LIN {X 0,Y 363.033,Z 812.389,A -85,B 0,C 180,E1 -13571.073,E2 -13571.073} C_VEL
LIN {X 0,Y 362.364,Z 824.695,A -85,B 0,C 180,E1 -13571.915,E2 -13571.915} C_VEL
LIN {X 0,Y 361.562,Z 836.062,A -85,B 0,C 180,E1 -13572.935,E2 -13572.935} C_VEL
LIN {X 0,Y 360.7,Z 845.735,A -85,B 0,C 180,E1 -13574.019,E2 -13574.019} C_VEL
LIN {X 0,Y 359.815,Z 854.935,A -85,B 0,C 180,E1 -13575.284,E2 -13575.284} C_VEL
LIN {X 0,Y 358.912,Z 863.313,A -85,B 0,C 180,E1 -13576.691,E2 -13576.691} C_VEL
LIN {X 0,Y 357.851,Z 871.446,A -85,B 0,C 180,E1 -13578.38,E2 -13578.38} C_VEL
LIN {X 0,Y 357.002,Z 878.309,A -85,B 0,C 180,E1 -13580.172,E2 -13580.172} C_VEL
LIN {X 0,Y 356.417,Z 883.932,A -85,B 0,C 180,E1 -13582.059,E2 -13582.059} C_VEL
LIN {X 0,Y 355.754,Z 887.827,A -85,B 0,C 180,E1 -13583.755,E2 -13583.755} C_VEL
LIN {X 0,Y 355.31,Z 890.694,A -85,B 0,C 180,E1 -13585.455,E2 -13585.455} C_VEL
LIN {X 0,Y 355.23,Z 892.053,A -85,B 0,C 180,E1 -13586.59,E2 -13586.59} C_VEL
LIN {X 0,Y 355.216,Z 893.011,A -85,B 0,C 180,E1 -13587.725,E2 -13587.725} C_VEL
LIN {X 0,Y 355.044,Z 893.855,A -85,B 0,C 180,E1 -13589.992,E2 -13589.992} C_VEL
LIN {X 0,Y 355.224,Z 893.093,A -85,B 0,C 180,E1 -13592.26,E2 -13592.26} C_VEL
LIN {X 0,Y 355.295,Z 890.863,A -85,B 0,C 180,E1 -13594.53,E2 -13594.53} C_VEL
LIN {X 0,Y 355.742,Z 888.05,A -85,B 0,C 180,E1 -13596.23,E2 -13596.23} C_VEL
LIN {X 0,Y 356.389,Z 884.226,A -85,B 0,C 180,E1 -13597.926,E2 -13597.926} C_VEL
LIN {X 0,Y 356.975,Z 878.755,A -85,B 0,C 180,E1 -13599.803,E2 -13599.803} C_VEL
LIN {X 0,Y 357.831,Z 871.946,A -85,B 0,C 180,E1 -13601.605,E2 -13601.605} C_VEL
LIN {X 0,Y 358.881,Z 863.92,A -85,B 0,C 180,E1 -13603.294,E2 -13603.294} C_VEL
LIN {X 0,Y 359.776,Z 855.705,A -85,B 0,C 180,E1 -13604.702,E2 -13604.702} C_VEL
LIN {X 0,Y 360.732,Z 845.541,A -85,B 0,C 180,E1 -13606.11,E2 -13606.11} C_VEL
LIN {X 0,Y 361.701,Z 835.452,A -85,B 0,C 180,E1 -13607.226,E2 -13607.226} C_VEL
LIN {X 0,Y 361.408,Z 832.183,A -85,B 0,C 180,E1 -13607.582,E2 -13607.582} C_VEL
LIN {X 0,Y 359.137,Z 827.141,A -85,B 0,C 180,E1 -13608.205,E2 -13608.205} C_VEL
LIN {X 0,Y 356.76,Z 821.949,A -85,B 0,C 180,E1 -13608.788,E2 -13608.788} C_VEL
LIN {X 0,Y 356.293,Z 818.404,A -85,B 0,C 180,E1 -13609.072,E2 -13609.072} C_VEL
LIN {X 0,Y 356.661,Z 805.402,A -85,B 0,C 180,E1 -13609.825,E2 -13609.825} C_VEL
LIN {X 0,Y 356.867,Z 793.247,A -85,B 0,C 180,E1 -13610.301,E2 -13610.301} C_VEL
LIN {X 0,Y 357.103,Z 760.469,A -85,B 0,C 180,E1 -13611.017,E2 -13611.017} C_VEL
LIN {X 0,Y 357.565,Z 732.208,A -85,B 0,C 180,E1 -13611.588,E2 -13611.588} C_VEL
LIN {X 0,Y 348.581,Z 711.641,A -85,B 0,C 180,E1 -13612.655,E2 -13612.655} C_VEL
LIN {X 0,Y 347.782,Z 709.155,A -85,B 0,C 180,E1 -13612.804,E2 -13612.804} C_VEL
LIN {X 0,Y 347.806,Z 709.153,A -85,B 0,C 180,E1 -13616.384,E2 -13616.384} C_VEL
LIN {X 0,Y 347.721,Z 709.167,A -85,B 0,C 180,E1 -13620.339,E2 -13620.339} C_VEL
LIN {X 0,Y 347.716,Z 709.168,A -85,B 0,C 180,E1 -13624.035,E2 -13624.035} C_VEL
LIN {X 0,Y 347.727,Z 709.161,A -85,B 0,C 180,E1 -13627.312,E2 -13627.312} C_VEL
LIN {X 0,Y 347.754,Z 709.168,A -85,B 0,C 180,E1 -13630.28,E2 -13630.28} C_VEL
LIN {X 0,Y 347.777,Z 709.158,A -85,B 0,C 180,E1 -13633.385,E2 -13633.385} C_VEL
LIN {X 0,Y 347.772,Z 709.156,A -85,B 0,C 180,E1 -13636.663,E2 -13636.663} C_VEL
LIN {X 0,Y 347.737,Z 709.167,A -85,B 0,C 180,E1 -13640.158,E2 -13640.158} C_VEL
LIN {X 0,Y 347.735,Z 709.169,A -85,B 0,C 180,E1 -13644.118,E2 -13644.118} C_VEL
LIN {X 0,Y 347.706,Z 709.173,A -85,B 0,C 180,E1 -13648.296,E2 -13648.296} C_VEL
LIN {X 0,Y 347.746,Z 709.157,A -85,B 0,C 180,E1 -13650.984,E2 -13650.984} C_VEL
LIN {X 0,Y 347.77,Z 709.163,A -85,B 0,C 180,E1 -13653.603,E2 -13653.603} C_VEL
LIN {X 0,Y 347.725,Z 709.163,A -85,B 0,C 180,E1 -13656.157,E2 -13656.157} C_VEL
LIN {X 0,Y 347.747,Z 709.167,A -85,B 0,C 180,E1 -13659.905,E2 -13659.905} C_VEL
LIN {X 0,Y 347.8,Z 709.152,A -85,B 0,C 180,E1 -13662.356,E2 -13662.356} C_VEL
LIN {X 0,Y 347.83,Z 709.157,A -85,B 0,C 180,E1 -13665.968,E2 -13665.968} C_VEL
LIN {X 0,Y 347.864,Z 709.142,A -85,B 0,C 180,E1 -13669.524,E2 -13669.524} C_VEL
LIN {X 0,Y 348.026,Z 709.136,A -85,B 0,C 180,E1 -13673.041,E2 -13673.041} C_VEL
LIN {X 0,Y 348.145,Z 709.117,A -85,B 0,C 180,E1 -13677.686,E2 -13677.686} C_VEL
LIN {X 0,Y 348.297,Z 709.1,A -85,B 0,C 180,E1 -13680,E2 -13680} C_VEL
LIN {X 0,Y 348.145,Z 709.112,A -85,B 0,C 180,E1 -13682.314,E2 -13682.314} C_VEL
LIN {X 0,Y 348.025,Z 709.138,A -85,B 0,C 180,E1 -13686.959,E2 -13686.959} C_VEL
LIN {X 0,Y 347.864,Z 709.148,A -85,B 0,C 180,E1 -13690.476,E2 -13690.476} C_VEL
LIN {X 0,Y 347.831,Z 709.155,A -85,B 0,C 180,E1 -13694.153,E2 -13694.153} C_VEL
LIN {X 0,Y 347.824,Z 709.156,A -85,B 0,C 180,E1 -13698.293,E2 -13698.293} C_VEL
LIN {X 0,Y 347.712,Z 709.164,A -85,B 0,C 180,E1 -13701.634,E2 -13701.634} C_VEL
LIN {X 0,Y 347.75,Z 709.163,A -85,B 0,C 180,E1 -13705.113,E2 -13705.113} C_VEL
LIN {X 0,Y 347.752,Z 709.166,A -85,B 0,C 180,E1 -13707.699,E2 -13707.699} C_VEL
LIN {X 0,Y 347.712,Z 709.165,A -85,B 0,C 180,E1 -13710.352,E2 -13710.352} C_VEL
LIN {X 0,Y 347.693,Z 709.171,A -85,B 0,C 180,E1 -13714.05,E2 -13714.05} C_VEL
LIN {X 0,Y 347.714,Z 709.168,A -85,B 0,C 180,E1 -13717.327,E2 -13717.327} C_VEL
LIN {X 0,Y 347.744,Z 709.161,A -85,B 0,C 180,E1 -13720.296,E2 -13720.296} C_VEL
LIN {X 0,Y 347.773,Z 709.164,A -85,B 0,C 180,E1 -13723.401,E2 -13723.401} C_VEL
LIN {X 0,Y 347.775,Z 709.16,A -85,B 0,C 180,E1 -13726.678,E2 -13726.678} C_VEL
LIN {X 0,Y 347.747,Z 709.166,A -85,B 0,C 180,E1 -13730.173,E2 -13730.173} C_VEL
LIN {X 0,Y 347.742,Z 709.238,A -85,B 0,C 180,E1 -13733.578,E2 -13733.578} C_VEL
LIN {X 0,Y 350.722,Z 720.967,A -85,B 0,C 180,E1 -13736.217,E2 -13736.217} C_VEL
LIN {X 0,Y 354.282,Z 737.106,A -85,B 0,C 180,E1 -13739.623,E2 -13739.623} C_VEL
LIN {X 0,Y 354.467,Z 740.581,A -85,B 0,C 180,E1 -13740.297,E2 -13740.297} C_VEL
LIN {X 0,Y 351.936,Z 764.083,A -85,B 0,C 180,E1 -13744.584,E2 -13744.584} C_VEL
LIN {X 0,Y 350.688,Z 776.95,A -85,B 0,C 180,E1 -13746.947,E2 -13746.947} C_VEL
LIN {X 0,Y 354.861,Z 812.933,A -85,B 0,C 180,E1 -13747.995,E2 -13747.995} C_VEL
LIN {X 0,Y 356.332,Z 830.994,A -85,B 0,C 180,E1 -13748.467,E2 -13748.467} C_VEL
LIN {X 0,Y 355.113,Z 888.22,A -85,B 0,C 180,E1 -13749.633,E2 -13749.633} C_VEL
LIN {X 0,Y 354.393,Z 902.169,A -85,B 0,C 180,E1 -13750.156,E2 -13750.156} C_VEL
LIN {X 0,Y 353.32,Z 914.672,A -85,B 0,C 180,E1 -13750.849,E2 -13750.849} C_VEL
LIN {X 0,Y 352.199,Z 925.867,A -85,B 0,C 180,E1 -13751.692,E2 -13751.692} C_VEL
LIN {X 0,Y 350.897,Z 937.551,A -85,B 0,C 180,E1 -13752.826,E2 -13752.826} C_VEL
LIN {X 0,Y 349.706,Z 948.114,A -85,B 0,C 180,E1 -13754.117,E2 -13754.117} C_VEL
LIN {X 0,Y 348.615,Z 957.541,A -85,B 0,C 180,E1 -13755.542,E2 -13755.542} C_VEL
LIN {X 0,Y 348.169,Z 963.316,A -85,B 0,C 180,E1 -13756.586,E2 -13756.586} C_VEL
LIN {X 0,Y 347.394,Z 971.527,A -85,B 0,C 180,E1 -13758.337,E2 -13758.337} C_VEL
LIN {X 0,Y 346.965,Z 978.154,A -85,B 0,C 180,E1 -13760.094,E2 -13760.094} C_VEL
LIN {X 0,Y 346.829,Z 983.454,A -85,B 0,C 180,E1 -13761.854,E2 -13761.854} C_VEL
LIN {X 0,Y 346.912,Z 987.231,A -85,B 0,C 180,E1 -13763.433,E2 -13763.433} C_VEL
LIN {X 0,Y 347.049,Z 990.682,A -85,B 0,C 180,E1 -13765.362,E2 -13765.362} C_VEL
LIN {X 0,Y 347.141,Z 992.149,A -85,B 0,C 180,E1 -13766.526,E2 -13766.526} C_VEL
LIN {X 0,Y 347.188,Z 993.192,A -85,B 0,C 180,E1 -13767.688,E2 -13767.688} C_VEL
LIN {X 0,Y 347.262,Z 993.833,A -85,B 0,C 180,E1 -13768.848,E2 -13768.848} C_VEL
LIN {X 0,Y 347.327,Z 994.062,A -85,B 0,C 180,E1 -13770.008,E2 -13770.008} C_VEL
LIN {X 0,Y 347.263,Z 993.822,A -85,B 0,C 180,E1 -13771.167,E2 -13771.167} C_VEL
LIN {X 0,Y 347.19,Z 993.173,A -85,B 0,C 180,E1 -13772.328,E2 -13772.328} C_VEL
LIN {X 0,Y 347.144,Z 992.122,A -85,B 0,C 180,E1 -13773.489,E2 -13773.489} C_VEL
LIN {X 0,Y 347.05,Z 990.643,A -85,B 0,C 180,E1 -13774.654,E2 -13774.654} C_VEL
LIN {X 0,Y 346.834,Z 986.62,A -85,B 0,C 180,E1 -13776.829,E2 -13776.829} C_VEL
LIN {X 0,Y 346.85,Z 981.728,A -85,B 0,C 180,E1 -13778.748,E2 -13778.748} C_VEL
LIN {X 0,Y 347.072,Z 975.988,A -85,B 0,C 180,E1 -13780.508,E2 -13780.508} C_VEL
LIN {X 0,Y 347.604,Z 968.877,A -85,B 0,C 180,E1 -13782.264,E2 -13782.264} C_VEL
LIN {X 0,Y 348.419,Z 960.016,A -85,B 0,C 180,E1 -13784.015,E2 -13784.015} C_VEL
LIN {X 0,Y 349.011,Z 954.446,A -85,B 0,C 180,E1 -13784.943,E2 -13784.943} C_VEL
LIN {X 0,Y 349.854,Z 945.728,A -85,B 0,C 180,E1 -13786.191,E2 -13786.191} C_VEL
LIN {X 0,Y 351.166,Z 934.653,A -85,B 0,C 180,E1 -13787.476,E2 -13787.476} C_VEL
LIN {X 0,Y 352.408,Z 923.864,A -85,B 0,C 180,E1 -13788.464,E2 -13788.464} C_VEL
LIN {X 0,Y 354.182,Z 906.155,A -85,B 0,C 180,E1 -13789.721,E2 -13789.721} C_VEL
LIN {X 0,Y 355.294,Z 895.091,A -85,B 0,C 180,E1 -13790.335,E2 -13790.335} C_VEL
LIN {X 0,Y 356.158,Z 883.683,A -85,B 0,C 180,E1 -13790.812,E2 -13790.812} C_VEL
LIN {X 0,Y 358.768,Z 828.38,A -85,B 0,C 180,E1 -13792.478,E2 -13792.478} C_VEL
LIN {X 0,Y 357.212,Z 800.501,A -85,B 0,C 180,E1 -13793.658,E2 -13793.658} C_VEL
LIN {X 0,Y 354.765,Z 779.754,A -85,B 0,C 180,E1 -13794.75,E2 -13794.75} C_VEL
LIN {X 0,Y 352.506,Z 764.919,A -85,B 0,C 180,E1 -13795.644,E2 -13795.644} C_VEL
LIN {X 0,Y 352.154,Z 761.628,A -85,B 0,C 180,E1 -13795.852,E2 -13795.852} C_VEL
LIN {X 0,Y 354.226,Z 742.379,A -85,B 0,C 180,E1 -13799.362,E2 -13799.362} C_VEL
LIN {X 0,Y 354.422,Z 738.666,A -85,B 0,C 180,E1 -13800.052,E2 -13800.052} C_VEL
LIN {X 0,Y 352.311,Z 727.989,A -85,B 0,C 180,E1 -13802.256,E2 -13802.256} C_VEL
LIN {X 0,Y 348.952,Z 714.025,A -85,B 0,C 180,E1 -13805.305,E2 -13805.305} C_VEL
LIN {X 0,Y 347.756,Z 709.154,A -85,B 0,C 180,E1 -13806.471,E2 -13806.471} C_VEL
LIN {X 0,Y 347.72,Z 709.172,A -85,B 0,C 180,E1 -13809.821,E2 -13809.821} C_VEL
LIN {X 0,Y 347.732,Z 709.172,A -85,B 0,C 180,E1 -13813.413,E2 -13813.413} C_VEL
LIN {X 0,Y 347.74,Z 709.166,A -85,B 0,C 180,E1 -13816.691,E2 -13816.691} C_VEL
LIN {X 0,Y 347.721,Z 709.17,A -85,B 0,C 180,E1 -13820.185,E2 -13820.185} C_VEL
LIN {X 0,Y 347.774,Z 709.162,A -85,B 0,C 180,E1 -13822.681,E2 -13822.681} C_VEL
LIN {X 0,Y 347.769,Z 709.164,A -85,B 0,C 180,E1 -13825.959,E2 -13825.959} C_VEL
LIN {X 0,Y 347.756,Z 709.167,A -85,B 0,C 180,E1 -13829.653,E2 -13829.653} C_VEL
LIN {X 0,Y 347.781,Z 709.266,A -85,B 0,C 180,E1 -13833.721,E2 -13833.721} C_VEL
LIN {X 0,Y 348.906,Z 712.205,A -85,B 0,C 180,E1 -13834.053,E2 -13834.053} C_VEL
LIN {X 0,Y 350.729,Z 714.546,A -85,B 0,C 180,E1 -13834.467,E2 -13834.467} C_VEL
LIN {X 0,Y 352.786,Z 717.784,A -85,B 0,C 180,E1 -13834.933,E2 -13834.933} C_VEL
LIN {X 0,Y 358.789,Z 728.477,A -85,B 0,C 180,E1 -13836.248,E2 -13836.248} C_VEL
LIN {X 0,Y 362.716,Z 736.606,A -85,B 0,C 180,E1 -13837.071,E2 -13837.071} C_VEL
LIN {X 0,Y 359.911,Z 789.103,A -85,B 0,C 180,E1 -13838.71,E2 -13838.71} C_VEL
LIN {X 0,Y 359.641,Z 803.34,A -85,B 0,C 180,E1 -13839.256,E2 -13839.256} C_VEL
LIN {X 0,Y 359.183,Z 814.12,A -85,B 0,C 180,E1 -13839.814,E2 -13839.814} C_VEL
LIN {X 0,Y 358.405,Z 827.548,A -85,B 0,C 180,E1 -13840.736,E2 -13840.736} C_VEL
LIN {X 0,Y 357.419,Z 839.218,A -85,B 0,C 180,E1 -13841.811,E2 -13841.811} C_VEL
LIN {X 0,Y 356.472,Z 848.007,A -85,B 0,C 180,E1 -13842.799,E2 -13842.799} C_VEL
LIN {X 0,Y 355.531,Z 856.33,A -85,B 0,C 180,E1 -13843.934,E2 -13843.934} C_VEL
LIN {X 0,Y 354.571,Z 863.373,A -85,B 0,C 180,E1 -13845.068,E2 -13845.068} C_VEL
LIN {X 0,Y 353.694,Z 869.433,A -85,B 0,C 180,E1 -13846.205,E2 -13846.205} C_VEL
LIN {X 0,Y 352.613,Z 876.291,A -85,B 0,C 180,E1 -13847.775,E2 -13847.775} C_VEL
LIN {X 0,Y 351.765,Z 880.973,A -85,B 0,C 180,E1 -13849.059,E2 -13849.059} C_VEL
LIN {X 0,Y 350.8,Z 885.918,A -85,B 0,C 180,E1 -13850.777,E2 -13850.777} C_VEL
LIN {X 0,Y 349.947,Z 889.668,A -85,B 0,C 180,E1 -13852.499,E2 -13852.499} C_VEL
LIN {X 0,Y 349.298,Z 892.334,A -85,B 0,C 180,E1 -13854.226,E2 -13854.226} C_VEL
LIN {X 0,Y 349.029,Z 893.606,A -85,B 0,C 180,E1 -13855.38,E2 -13855.38} C_VEL
LIN {X 0,Y 348.461,Z 894.672,A -85,B 0,C 180,E1 -13857.688,E2 -13857.688} C_VEL
LIN {X 0,Y 348.268,Z 894.566,A -85,B 0,C 180,E1 -13858.844,E2 -13858.844} C_VEL
LIN {X 0,Y 348.031,Z 894.004,A -85,B 0,C 180,E1 -13860,E2 -13860} C_VEL
LIN {X 0,Y 347.875,Z 891.603,A -85,B 0,C 180,E1 -13862.316,E2 -13862.316} C_VEL
LIN {X 0,Y 347.823,Z 888.615,A -85,B 0,C 180,E1 -13864.055,E2 -13864.055} C_VEL
LIN {X 0,Y 348.192,Z 884.49,A -85,B 0,C 180,E1 -13865.792,E2 -13865.792} C_VEL
LIN {X 0,Y 348.488,Z 879.178,A -85,B 0,C 180,E1 -13867.532,E2 -13867.532} C_VEL
LIN {X 0,Y 348.81,Z 873.146,A -85,B 0,C 180,E1 -13869.127,E2 -13869.127} C_VEL
LIN {X 0,Y 349.155,Z 867.226,A -85,B 0,C 180,E1 -13870.437,E2 -13870.437} C_VEL
LIN {X 0,Y 349.647,Z 859.367,A -85,B 0,C 180,E1 -13871.89,E2 -13871.89} C_VEL
LIN {X 0,Y 350.099,Z 850.899,A -85,B 0,C 180,E1 -13873.2,E2 -13873.2} C_VEL
LIN {X 0,Y 350.606,Z 841.924,A -85,B 0,C 180,E1 -13874.363,E2 -13874.363} C_VEL
LIN {X 0,Y 351.081,Z 834.019,A -85,B 0,C 180,E1 -13875.233,E2 -13875.233} C_VEL
LIN {X 0,Y 351.558,Z 823.838,A -85,B 0,C 180,E1 -13876.169,E2 -13876.169} C_VEL
LIN {X 0,Y 351.952,Z 813.596,A -85,B 0,C 180,E1 -13876.935,E2 -13876.935} C_VEL
LIN {X 0,Y 352.228,Z 803.005,A -85,B 0,C 180,E1 -13877.565,E2 -13877.565} C_VEL
LIN {X 0,Y 352.457,Z 792.447,A -85,B 0,C 180,E1 -13878.041,E2 -13878.041} C_VEL
LIN {X 0,Y 352.627,Z 778.382,A -85,B 0,C 180,E1 -13878.483,E2 -13878.483} C_VEL
LIN {X 0,Y 353.651,Z 727.317,A -85,B 0,C 180,E1 -13879.826,E2 -13879.826} C_VEL
LIN {X 0,Y 347.832,Z 709.16,A -85,B 0,C 180,E1 -13880.594,E2 -13880.594} C_VEL
LIN {X 0,Y 347.824,Z 709.16,A -85,B 0,C 180,E1 -13884.588,E2 -13884.588} C_VEL
LIN {X 0,Y 347.757,Z 709.162,A -85,B 0,C 180,E1 -13887.699,E2 -13887.699} C_VEL
LIN {X 0,Y 347.757,Z 709.166,A -85,B 0,C 180,E1 -13890.347,E2 -13890.347} C_VEL
LIN {X 0,Y 347.77,Z 709.161,A -85,B 0,C 180,E1 -13894.041,E2 -13894.041} C_VEL
LIN {X 0,Y 347.775,Z 709.163,A -85,B 0,C 180,E1 -13897.319,E2 -13897.319} C_VEL
LIN {X 0,Y 347.717,Z 709.168,A -85,B 0,C 180,E1 -13900.299,E2 -13900.299} C_VEL
LIN {X 0,Y 347.741,Z 709.164,A -85,B 0,C 180,E1 -13903.406,E2 -13903.406} C_VEL
LIN {X 0,Y 347.743,Z 709.163,A -85,B 0,C 180,E1 -13906.684,E2 -13906.684} C_VEL
LIN {X 0,Y 347.721,Z 709.164,A -85,B 0,C 180,E1 -13910.179,E2 -13910.179} C_VEL
LIN {X 0,Y 347.773,Z 709.16,A -85,B 0,C 180,E1 -13912.674,E2 -13912.674} C_VEL
LIN {X 0,Y 347.767,Z 709.159,A -85,B 0,C 180,E1 -13915.952,E2 -13915.952} C_VEL
LIN {X 0,Y 347.744,Z 709.165,A -85,B 0,C 180,E1 -13919.645,E2 -13919.645} C_VEL
LIN {X 0,Y 347.748,Z 709.166,A -85,B 0,C 180,E1 -13923.594,E2 -13923.594} C_VEL
LIN {X 0,Y 347.799,Z 709.163,A -85,B 0,C 180,E1 -13927.337,E2 -13927.337} C_VEL
LIN {X 0,Y 348.822,Z 712.011,A -85,B 0,C 180,E1 -13927.479,E2 -13927.479} C_VEL
LIN {X 0,Y 357.48,Z 732.053,A -85,B 0,C 180,E1 -13928.51,E2 -13928.51} C_VEL
LIN {X 0,Y 356.849,Z 788.301,A -85,B 0,C 180,E1 -13929.67,E2 -13929.67} C_VEL
LIN {X 0,Y 356.776,Z 801.73,A -85,B 0,C 180,E1 -13930.117,E2 -13930.117} C_VEL
LIN {X 0,Y 356.395,Z 813.4,A -85,B 0,C 180,E1 -13930.706,E2 -13930.706} C_VEL
LIN {X 0,Y 355.69,Z 825.704,A -85,B 0,C 180,E1 -13931.564,E2 -13931.564} C_VEL
LIN {X 0,Y 354.849,Z 837.07,A -85,B 0,C 180,E1 -13932.602,E2 -13932.602} C_VEL
LIN {X 0,Y 353.949,Z 846.742,A -85,B 0,C 180,E1 -13933.705,E2 -13933.705} C_VEL
LIN {X 0,Y 353.023,Z 855.941,A -85,B 0,C 180,E1 -13934.994,E2 -13934.994} C_VEL
LIN {X 0,Y 352.076,Z 864.318,A -85,B 0,C 180,E1 -13936.428,E2 -13936.428} C_VEL
LIN {X 0,Y 350.971,Z 872.451,A -85,B 0,C 180,E1 -13938.149,E2 -13938.149} C_VEL
LIN {X 0,Y 350.079,Z 879.313,A -85,B 0,C 180,E1 -13939.976,E2 -13939.976} C_VEL
LIN {X 0,Y 349.459,Z 884.936,A -85,B 0,C 180,E1 -13941.9,E2 -13941.9} C_VEL
LIN {X 0,Y 348.77,Z 888.831,A -85,B 0,C 180,E1 -13943.63,E2 -13943.63} C_VEL
LIN {X 0,Y 348.304,Z 891.698,A -85,B 0,C 180,E1 -13945.363,E2 -13945.363} C_VEL
LIN {X 0,Y 348.215,Z 893.056,A -85,B 0,C 180,E1 -13946.521,E2 -13946.521} C_VEL
LIN {X 0,Y 348.196,Z 894.014,A -85,B 0,C 180,E1 -13947.679,E2 -13947.679} C_VEL
LIN {X 0,Y 348.017,Z 894.857,A -85,B 0,C 180,E1 -13949.992,E2 -13949.992} C_VEL
LIN {X 0,Y 348.203,Z 894.095,A -85,B 0,C 180,E1 -13952.306,E2 -13952.306} C_VEL
LIN {X 0,Y 348.288,Z 891.865,A -85,B 0,C 180,E1 -13954.622,E2 -13954.622} C_VEL
LIN {X 0,Y 348.758,Z 889.052,A -85,B 0,C 180,E1 -13956.355,E2 -13956.355} C_VEL
LIN {X 0,Y 349.433,Z 885.227,A -85,B 0,C 180,E1 -13958.085,E2 -13958.085} C_VEL
LIN {X 0,Y 350.052,Z 879.756,A -85,B 0,C 180,E1 -13959.999,E2 -13959.999} C_VEL
LIN {X 0,Y 350.95,Z 872.946,A -85,B 0,C 180,E1 -13961.836,E2 -13961.836} C_VEL
LIN {X 0,Y 352.047,Z 864.92,A -85,B 0,C 180,E1 -13963.557,E2 -13963.557} C_VEL
LIN {X 0,Y 352.982,Z 856.705,A -85,B 0,C 180,E1 -13964.992,E2 -13964.992} C_VEL
LIN {X 0,Y 353.987,Z 846.54,A -85,B 0,C 180,E1 -13966.425,E2 -13966.425} C_VEL
LIN {X 0,Y 355.045,Z 836.075,A -85,B 0,C 180,E1 -13967.599,E2 -13967.599} C_VEL
LIN {X 0,Y 355.858,Z 824.814,A -85,B 0,C 180,E1 -13968.609,E2 -13968.609} C_VEL
LIN {X 0,Y 356.293,Z 818.404,A -85,B 0,C 180,E1 -13969.072,E2 -13969.072} C_VEL
LIN {X 0,Y 355.976,Z 812.981,A -85,B 0,C 180,E1 -13969.452,E2 -13969.452} C_VEL
LIN {X 0,Y 352.445,Z 800.677,A -85,B 0,C 180,E1 -13970.321,E2 -13970.321} C_VEL
LIN {X 0,Y 350.683,Z 793.351,A -85,B 0,C 180,E1 -13970.703,E2 -13970.703} C_VEL
LIN {X 0,Y 350.349,Z 789.515,A -85,B 0,C 180,E1 -13970.827,E2 -13970.827} C_VEL
LIN {X 0,Y 350.766,Z 749.924,A -85,B 0,C 180,E1 -13971.665,E2 -13971.665} C_VEL
LIN {X 0,Y 351.042,Z 733.993,A -85,B 0,C 180,E1 -13971.992,E2 -13971.992} C_VEL
LIN {X 0,Y 341.602,Z 712.634,A -85,B 0,C 180,E1 -13973.146,E2 -13973.146} C_VEL
LIN {X 0,Y 340.745,Z 710.035,A -85,B 0,C 180,E1 -13973.302,E2 -13973.302} C_VEL
LIN {X 0,Y 340.779,Z 710.033,A -85,B 0,C 180,E1 -13976.971,E2 -13976.971} C_VEL
LIN {X 0,Y 340.669,Z 710.05,A -85,B 0,C 180,E1 -13981.036,E2 -13981.036} C_VEL
LIN {X 0,Y 340.685,Z 710.049,A -85,B 0,C 180,E1 -13985.27,E2 -13985.27} C_VEL
LIN {X 0,Y 340.676,Z 710.03,A -85,B 0,C 180,E1 -13988.378,E2 -13988.378} C_VEL
LIN {X 0,Y 340.685,Z 710.052,A -85,B 0,C 180,E1 -13991.296,E2 -13991.296} C_VEL
LIN {X 0,Y 340.738,Z 710.023,A -85,B 0,C 180,E1 -13994.515,E2 -13994.515} C_VEL
LIN {X 0,Y 340.705,Z 710.046,A -85,B 0,C 180,E1 -13997.937,E2 -13997.937} C_VEL
LIN {X 0,Y 340.684,Z 710.045,A -85,B 0,C 180,E1 -14000.245,E2 -14000.245} C_VEL
LIN {X 0,Y 340.658,Z 710.052,A -85,B 0,C 180,E1 -14003.553,E2 -14003.553} C_VEL
LIN {X 0,Y 340.64,Z 710.048,A -85,B 0,C 180,E1 -14006.147,E2 -14006.147} C_VEL
LIN {X 0,Y 340.717,Z 710.035,A -85,B 0,C 180,E1 -14010.327,E2 -14010.327} C_VEL
LIN {X 0,Y 340.744,Z 710.037,A -85,B 0,C 180,E1 -14013.015,E2 -14013.015} C_VEL
LIN {X 0,Y 340.665,Z 710.043,A -85,B 0,C 180,E1 -14016.922,E2 -14016.922} C_VEL
LIN {X 0,Y 340.725,Z 710.038,A -85,B 0,C 180,E1 -14020.73,E2 -14020.73} C_VEL
LIN {X 0,Y 340.72,Z 710.034,A -85,B 0,C 180,E1 -14023.215,E2 -14023.215} C_VEL
LIN {X 0,Y 340.778,Z 710.035,A -85,B 0,C 180,E1 -14026.888,E2 -14026.888} C_VEL
LIN {X 0,Y 340.859,Z 710.019,A -85,B 0,C 180,E1 -14030.506,E2 -14030.506} C_VEL
LIN {X 0,Y 340.993,Z 710.014,A -85,B 0,C 180,E1 -14032.896,E2 -14032.896} C_VEL
LIN {X 0,Y 341.108,Z 709.994,A -85,B 0,C 180,E1 -14037.638,E2 -14037.638} C_VEL
LIN {X 0,Y 341.246,Z 709.979,A -85,B 0,C 180,E1 -14040,E2 -14040} C_VEL
LIN {X 0,Y 341.108,Z 709.988,A -85,B 0,C 180,E1 -14042.362,E2 -14042.362} C_VEL
LIN {X 0,Y 340.993,Z 710.012,A -85,B 0,C 180,E1 -14047.103,E2 -14047.103} C_VEL
LIN {X 0,Y 340.806,Z 710.028,A -85,B 0,C 180,E1 -14050.696,E2 -14050.696} C_VEL
LIN {X 0,Y 340.796,Z 710.031,A -85,B 0,C 180,E1 -14054.328,E2 -14054.328} C_VEL
LIN {X 0,Y 340.771,Z 710.034,A -85,B 0,C 180,E1 -14058.469,E2 -14058.469} C_VEL
LIN {X 0,Y 340.659,Z 710.045,A -85,B 0,C 180,E1 -14061.848,E2 -14061.848} C_VEL
LIN {X 0,Y 340.711,Z 710.037,A -85,B 0,C 180,E1 -14065.669,E2 -14065.669} C_VEL
LIN {X 0,Y 340.682,Z 710.046,A -85,B 0,C 180,E1 -14068.325,E2 -14068.325} C_VEL
LIN {X 0,Y 340.658,Z 710.044,A -85,B 0,C 180,E1 -14071.049,E2 -14071.049} C_VEL
LIN {X 0,Y 340.664,Z 710.047,A -85,B 0,C 180,E1 -14075.285,E2 -14075.285} C_VEL
LIN {X 0,Y 340.663,Z 710.034,A -85,B 0,C 180,E1 -14078.394,E2 -14078.394} C_VEL
LIN {X 0,Y 340.677,Z 710.048,A -85,B 0,C 180,E1 -14081.311,E2 -14081.311} C_VEL
LIN {X 0,Y 340.736,Z 710.041,A -85,B 0,C 180,E1 -14084.53,E2 -14084.53} C_VEL
LIN {X 0,Y 340.71,Z 710.036,A -85,B 0,C 180,E1 -14087.953,E2 -14087.953} C_VEL
LIN {X 0,Y 340.695,Z 710.043,A -85,B 0,C 180,E1 -14090.26,E2 -14090.26} C_VEL
LIN {X 0,Y 340.698,Z 710.136,A -85,B 0,C 180,E1 -14093.109,E2 -14093.109} C_VEL
LIN {X 0,Y 344.101,Z 723.516,A -85,B 0,C 180,E1 -14096.194,E2 -14096.194} C_VEL
LIN {X 0,Y 347.263,Z 737.936,A -85,B 0,C 180,E1 -14099.307,E2 -14099.307} C_VEL
LIN {X 0,Y 347.647,Z 740.989,A -85,B 0,C 180,E1 -14099.929,E2 -14099.929} C_VEL
LIN {X 0,Y 345.199,Z 763.104,A -85,B 0,C 180,E1 -14104.058,E2 -14104.058} C_VEL
LIN {X 0,Y 343.868,Z 776.212,A -85,B 0,C 180,E1 -14106.478,E2 -14106.478} C_VEL
LIN {X 0,Y 347.914,Z 810.535,A -85,B 0,C 180,E1 -14107.502,E2 -14107.502} C_VEL
LIN {X 0,Y 349.706,Z 831.274,A -85,B 0,C 180,E1 -14108.065,E2 -14108.065} C_VEL
LIN {X 0,Y 348.435,Z 887.216,A -85,B 0,C 180,E1 -14109.224,E2 -14109.224} C_VEL
LIN {X 0,Y 347.781,Z 900.401,A -85,B 0,C 180,E1 -14109.724,E2 -14109.724} C_VEL
LIN {X 0,Y 346.647,Z 913.669,A -85,B 0,C 180,E1 -14110.466,E2 -14110.466} C_VEL
LIN {X 0,Y 345.443,Z 924.856,A -85,B 0,C 180,E1 -14111.32,E2 -14111.32} C_VEL
LIN {X 0,Y 344.084,Z 936.537,A -85,B 0,C 180,E1 -14112.475,E2 -14112.475} C_VEL
LIN {X 0,Y 342.778,Z 947.088,A -85,B 0,C 180,E1 -14113.788,E2 -14113.788} C_VEL
LIN {X 0,Y 341.778,Z 955.796,A -85,B 0,C 180,E1 -14115.12,E2 -14115.12} C_VEL
LIN {X 0,Y 341.247,Z 962.302,A -85,B 0,C 180,E1 -14116.309,E2 -14116.309} C_VEL
LIN {X 0,Y 340.394,Z 970.509,A -85,B 0,C 180,E1 -14118.093,E2 -14118.093} C_VEL
LIN {X 0,Y 339.918,Z 977.134,A -85,B 0,C 180,E1 -14119.887,E2 -14119.887} C_VEL
LIN {X 0,Y 339.758,Z 982.435,A -85,B 0,C 180,E1 -14121.683,E2 -14121.683} C_VEL
LIN {X 0,Y 339.829,Z 985.719,A -85,B 0,C 180,E1 -14123.068,E2 -14123.068} C_VEL
LIN {X 0,Y 339.992,Z 989.672,A -85,B 0,C 180,E1 -14125.265,E2 -14125.265} C_VEL
LIN {X 0,Y 340.096,Z 991.142,A -85,B 0,C 180,E1 -14126.454,E2 -14126.454} C_VEL
LIN {X 0,Y 340.145,Z 992.187,A -85,B 0,C 180,E1 -14127.64,E2 -14127.64} C_VEL
LIN {X 0,Y 340.226,Z 992.829,A -85,B 0,C 180,E1 -14128.824,E2 -14128.824} C_VEL
LIN {X 0,Y 340.297,Z 993.059,A -85,B 0,C 180,E1 -14130.008,E2 -14130.008} C_VEL
LIN {X 0,Y 340.226,Z 992.818,A -85,B 0,C 180,E1 -14131.191,E2 -14131.191} C_VEL
LIN {X 0,Y 340.147,Z 992.167,A -85,B 0,C 180,E1 -14132.376,E2 -14132.376} C_VEL
LIN {X 0,Y 340.099,Z 991.114,A -85,B 0,C 180,E1 -14133.562,E2 -14133.562} C_VEL
LIN {X 0,Y 339.991,Z 989.632,A -85,B 0,C 180,E1 -14134.75,E2 -14134.75} C_VEL
LIN {X 0,Y 339.777,Z 985.85,A -85,B 0,C 180,E1 -14136.859,E2 -14136.859} C_VEL
LIN {X 0,Y 339.799,Z 980.709,A -85,B 0,C 180,E1 -14138.931,E2 -14138.931} C_VEL
LIN {X 0,Y 340.012,Z 974.962,A -85,B 0,C 180,E1 -14140.728,E2 -14140.728} C_VEL
LIN {X 0,Y 340.597,Z 967.852,A -85,B 0,C 180,E1 -14142.52,E2 -14142.52} C_VEL
LIN {X 0,Y 341.342,Z 960.629,A -85,B 0,C 180,E1 -14144.007,E2 -14144.007} C_VEL
LIN {X 0,Y 341.669,Z 956.525,A -85,B 0,C 180,E1 -14144.746,E2 -14144.746} C_VEL
LIN {X 0,Y 342.727,Z 947.967,A -85,B 0,C 180,E1 -14146.078,E2 -14146.078} C_VEL
LIN {X 0,Y 343.914,Z 937.592,A -85,B 0,C 180,E1 -14147.396,E2 -14147.396} C_VEL
LIN {X 0,Y 345.657,Z 923.215,A -85,B 0,C 180,E1 -14148.838,E2 -14148.838} C_VEL
LIN {X 0,Y 346.914,Z 913.267,A -85,B 0,C 180,E1 -14149.689,E2 -14149.689} C_VEL
LIN {X 0,Y 348.062,Z 903.107,A -85,B 0,C 180,E1 -14150.391,E2 -14150.391} C_VEL
LIN {X 0,Y 349.241,Z 891.716,A -85,B 0,C 180,E1 -14151.012,E2 -14151.012} C_VEL
LIN {X 0,Y 350.096,Z 880.865,A -85,B 0,C 180,E1 -14151.459,E2 -14151.459} C_VEL
LIN {X 0,Y 352.68,Z 828.91,A -85,B 0,C 180,E1 -14153.081,E2 -14153.081} C_VEL
LIN {X 0,Y 351.318,Z 801.407,A -85,B 0,C 180,E1 -14154.3,E2 -14154.3} C_VEL
LIN {X 0,Y 349.158,Z 781.767,A -85,B 0,C 180,E1 -14155.378,E2 -14155.378} C_VEL
LIN {X 0,Y 346.526,Z 763.396,A -85,B 0,C 180,E1 -14156.538,E2 -14156.538} C_VEL
LIN {X 0,Y 345.726,Z 757.568,A -85,B 0,C 180,E1 -14156.963,E2 -14156.963} C_VEL
LIN {X 0,Y 347.567,Z 740.712,A -85,B 0,C 180,E1 -14160.113,E2 -14160.113} C_VEL
LIN {X 0,Y 345.641,Z 730.447,A -85,B 0,C 180,E1 -14162.266,E2 -14162.266} C_VEL
LIN {X 0,Y 342.372,Z 716.624,A -85,B 0,C 180,E1 -14165.348,E2 -14165.348} C_VEL
LIN {X 0,Y 340.716,Z 710.035,A -85,B 0,C 180,E1 -14166.932,E2 -14166.932} C_VEL
LIN {X 0,Y 340.669,Z 710.048,A -85,B 0,C 180,E1 -14170.243,E2 -14170.243} C_VEL
LIN {X 0,Y 340.662,Z 710.05,A -85,B 0,C 180,E1 -14173.775,E2 -14173.775} C_VEL
LIN {X 0,Y 340.684,Z 710.047,A -85,B 0,C 180,E1 -14177.097,E2 -14177.097} C_VEL
LIN {X 0,Y 340.675,Z 710.047,A -85,B 0,C 180,E1 -14180.244,E2 -14180.244} C_VEL
LIN {X 0,Y 340.727,Z 710.045,A -85,B 0,C 180,E1 -14183.563,E2 -14183.563} C_VEL
LIN {X 0,Y 340.711,Z 710.042,A -85,B 0,C 180,E1 -14186.155,E2 -14186.155} C_VEL
LIN {X 0,Y 340.74,Z 710.04,A -85,B 0,C 180,E1 -14190.038,E2 -14190.038} C_VEL
LIN {X 0,Y 340.754,Z 710.246,A -85,B 0,C 180,E1 -14192.492,E2 -14192.492} C_VEL
LIN {X 0,Y 341.762,Z 712.908,A -85,B 0,C 180,E1 -14192.83,E2 -14192.83} C_VEL
LIN {X 0,Y 343.792,Z 715.402,A -85,B 0,C 180,E1 -14193.347,E2 -14193.347} C_VEL
LIN {X 0,Y 345.708,Z 718.547,A -85,B 0,C 180,E1 -14193.83,E2 -14193.83} C_VEL
LIN {X 0,Y 350.832,Z 726.883,A -85,B 0,C 180,E1 -14195.057,E2 -14195.057} C_VEL
LIN {X 0,Y 356.547,Z 738.013,A -85,B 0,C 180,E1 -14196.353,E2 -14196.353} C_VEL
LIN {X 0,Y 356.969,Z 739.093,A -85,B 0,C 180,E1 -14196.452,E2 -14196.452} C_VEL
LIN {X 0,Y 353.976,Z 790.114,A -85,B 0,C 180,E1 -14198.106,E2 -14198.106} C_VEL
LIN {X 0,Y 353.666,Z 804.276,A -85,B 0,C 180,E1 -14198.66,E2 -14198.66} C_VEL
LIN {X 0,Y 353.269,Z 813.946,A -85,B 0,C 180,E1 -14199.159,E2 -14199.159} C_VEL
LIN {X 0,Y 352.675,Z 824.025,A -85,B 0,C 180,E1 -14199.827,E2 -14199.827} C_VEL
LIN {X 0,Y 352.002,Z 832.285,A -85,B 0,C 180,E1 -14200.493,E2 -14200.493} C_VEL
LIN {X 0,Y 351.207,Z 840.853,A -85,B 0,C 180,E1 -14201.326,E2 -14201.326} C_VEL
LIN {X 0,Y 350.173,Z 849.534,A -85,B 0,C 180,E1 -14202.328,E2 -14202.328} C_VEL
LIN {X 0,Y 349.315,Z 856.902,A -85,B 0,C 180,E1 -14203.339,E2 -14203.339} C_VEL
LIN {X 0,Y 348.316,Z 864.07,A -85,B 0,C 180,E1 -14204.494,E2 -14204.494} C_VEL
LIN {X 0,Y 347.104,Z 871.503,A -85,B 0,C 180,E1 -14205.938,E2 -14205.938} C_VEL
LIN {X 0,Y 346.031,Z 877.693,A -85,B 0,C 180,E1 -14207.407,E2 -14207.407} C_VEL
LIN {X 0,Y 345.026,Z 882.722,A -85,B 0,C 180,E1 -14208.842,E2 -14208.842} C_VEL
LIN {X 0,Y 344.412,Z 886.162,A -85,B 0,C 180,E1 -14210.012,E2 -14210.012} C_VEL
LIN {X 0,Y 343.374,Z 890.208,A -85,B 0,C 180,E1 -14211.763,E2 -14211.763} C_VEL
LIN {X 0,Y 342.765,Z 892.224,A -85,B 0,C 180,E1 -14212.933,E2 -14212.933} C_VEL
LIN {X 0,Y 342.087,Z 894.914,A -85,B 0,C 180,E1 -14215.286,E2 -14215.286} C_VEL
LIN {X 0,Y 341.483,Z 895.869,A -85,B 0,C 180,E1 -14217.641,E2 -14217.641} C_VEL
LIN {X 0,Y 341.283,Z 895.663,A -85,B 0,C 180,E1 -14218.82,E2 -14218.82} C_VEL
LIN {X 0,Y 341.008,Z 895.042,A -85,B 0,C 180,E1 -14220,E2 -14220} C_VEL
LIN {X 0,Y 340.848,Z 892.447,A -85,B 0,C 180,E1 -14222.364,E2 -14222.364} C_VEL
LIN {X 0,Y 340.8,Z 889.32,A -85,B 0,C 180,E1 -14224.139,E2 -14224.139} C_VEL
LIN {X 0,Y 341.15,Z 885.066,A -85,B 0,C 180,E1 -14225.912,E2 -14225.912} C_VEL
LIN {X 0,Y 341.418,Z 880.654,A -85,B 0,C 180,E1 -14227.392,E2 -14227.392} C_VEL
LIN {X 0,Y 341.696,Z 875.52,A -85,B 0,C 180,E1 -14228.823,E2 -14228.823} C_VEL
LIN {X 0,Y 342.054,Z 868.867,A -85,B 0,C 180,E1 -14230.357,E2 -14230.357} C_VEL
LIN {X 0,Y 342.549,Z 861.092,A -85,B 0,C 180,E1 -14231.839,E2 -14231.839} C_VEL
LIN {X 0,Y 343.02,Z 852.723,A -85,B 0,C 180,E1 -14233.176,E2 -14233.176} C_VEL
LIN {X 0,Y 343.501,Z 843.871,A -85,B 0,C 180,E1 -14234.364,E2 -14234.364} C_VEL
LIN {X 0,Y 344.084,Z 834.655,A -85,B 0,C 180,E1 -14235.398,E2 -14235.398} C_VEL
LIN {X 0,Y 344.508,Z 825.929,A -85,B 0,C 180,E1 -14236.226,E2 -14236.226} C_VEL
LIN {X 0,Y 344.962,Z 814.467,A -85,B 0,C 180,E1 -14237.106,E2 -14237.106} C_VEL
LIN {X 0,Y 345.242,Z 803.989,A -85,B 0,C 180,E1 -14237.741,E2 -14237.741} C_VEL
LIN {X 0,Y 345.489,Z 793.454,A -85,B 0,C 180,E1 -14238.226,E2 -14238.226} C_VEL
LIN {X 0,Y 345.635,Z 779.445,A -85,B 0,C 180,E1 -14238.678,E2 -14238.678} C_VEL
LIN {X 0,Y 346.676,Z 728.505,A -85,B 0,C 180,E1 -14240.055,E2 -14240.055} C_VEL
LIN {X 0,Y 340.763,Z 710.04,A -85,B 0,C 180,E1 -14240.839,E2 -14240.839} C_VEL
LIN {X 0,Y 340.759,Z 710.039,A -85,B 0,C 180,E1 -14244.831,E2 -14244.831} C_VEL
LIN {X 0,Y 340.704,Z 710.042,A -85,B 0,C 180,E1 -14248.323,E2 -14248.323} C_VEL
LIN {X 0,Y 340.712,Z 710.045,A -85,B 0,C 180,E1 -14251.043,E2 -14251.043} C_VEL
LIN {X 0,Y 340.736,Z 710.039,A -85,B 0,C 180,E1 -14255.277,E2 -14255.277} C_VEL
LIN {X 0,Y 340.714,Z 710.041,A -85,B 0,C 180,E1 -14258.379,E2 -14258.379} C_VEL
LIN {X 0,Y 340.711,Z 710.038,A -85,B 0,C 180,E1 -14262.04,E2 -14262.04} C_VEL
LIN {X 0,Y 340.67,Z 710.043,A -85,B 0,C 180,E1 -14266.224,E2 -14266.224} C_VEL
LIN {X 0,Y 340.688,Z 710.043,A -85,B 0,C 180,E1 -14268.684,E2 -14268.684} C_VEL
LIN {X 0,Y 340.738,Z 710.035,A -85,B 0,C 180,E1 -14271.766,E2 -14271.766} C_VEL
LIN {X 0,Y 340.741,Z 710.037,A -85,B 0,C 180,E1 -14275.592,E2 -14275.592} C_VEL
LIN {X 0,Y 340.699,Z 710.042,A -85,B 0,C 180,E1 -14278.949,E2 -14278.949} C_VEL
LIN {X 0,Y 340.725,Z 710.041,A -85,B 0,C 180,E1 -14283.006,E2 -14283.006} C_VEL
LIN {X 0,Y 340.735,Z 710.041,A -85,B 0,C 180,E1 -14286.827,E2 -14286.827} C_VEL
LIN {X 0,Y 341.729,Z 712.85,A -85,B 0,C 180,E1 -14286.979,E2 -14286.979} C_VEL
LIN {X 0,Y 350.762,Z 733.385,A -85,B 0,C 180,E1 -14288.084,E2 -14288.084} C_VEL
LIN {X 0,Y 350.973,Z 737.009,A -85,B 0,C 180,E1 -14288.177,E2 -14288.177} C_VEL
LIN {X 0,Y 350.253,Z 788.436,A -85,B 0,C 180,E1 -14289.247,E2 -14289.247} C_VEL
LIN {X 0,Y 350.169,Z 802.04,A -85,B 0,C 180,E1 -14289.696,E2 -14289.696} C_VEL
LIN {X 0,Y 349.767,Z 814.412,A -85,B 0,C 180,E1 -14290.326,E2 -14290.326} C_VEL
LIN {X 0,Y 349.03,Z 826.713,A -85,B 0,C 180,E1 -14291.199,E2 -14291.199} C_VEL
LIN {X 0,Y 348.15,Z 838.077,A -85,B 0,C 180,E1 -14292.256,E2 -14292.256} C_VEL
LIN {X 0,Y 347.209,Z 847.748,A -85,B 0,C 180,E1 -14293.38,E2 -14293.38} C_VEL
LIN {X 0,Y 346.24,Z 856.947,A -85,B 0,C 180,E1 -14294.693,E2 -14294.693} C_VEL
LIN {X 0,Y 345.249,Z 865.323,A -85,B 0,C 180,E1 -14296.154,E2 -14296.154} C_VEL
LIN {X 0,Y 344.096,Z 873.456,A -85,B 0,C 180,E1 -14297.909,E2 -14297.909} C_VEL
LIN {X 0,Y 343.161,Z 880.318,A -85,B 0,C 180,E1 -14299.771,E2 -14299.771} C_VEL
LIN {X 0,Y 342.504,Z 885.94,A -85,B 0,C 180,E1 -14301.734,E2 -14301.734} C_VEL
LIN {X 0,Y 341.787,Z 889.834,A -85,B 0,C 180,E1 -14303.499,E2 -14303.499} C_VEL
LIN {X 0,Y 341.299,Z 892.701,A -85,B 0,C 180,E1 -14305.268,E2 -14305.268} C_VEL
LIN {X 0,Y 341.2,Z 894.059,A -85,B 0,C 180,E1 -14306.45,E2 -14306.45} C_VEL
LIN {X 0,Y 341.177,Z 895.017,A -85,B 0,C 180,E1 -14307.631,E2 -14307.631} C_VEL
LIN {X 0,Y 340.991,Z 895.859,A -85,B 0,C 180,E1 -14309.992,E2 -14309.992} C_VEL
LIN {X 0,Y 341.182,Z 895.097,A -85,B 0,C 180,E1 -14312.353,E2 -14312.353} C_VEL
LIN {X 0,Y 341.283,Z 892.867,A -85,B 0,C 180,E1 -14314.717,E2 -14314.717} C_VEL
LIN {X 0,Y 341.775,Z 890.054,A -85,B 0,C 180,E1 -14316.486,E2 -14316.486} C_VEL
LIN {X 0,Y 342.479,Z 886.228,A -85,B 0,C 180,E1 -14318.25,E2 -14318.25} C_VEL
LIN {X 0,Y 343.133,Z 880.757,A -85,B 0,C 180,E1 -14320.203,E2 -14320.203} C_VEL
LIN {X 0,Y 344.075,Z 873.947,A -85,B 0,C 180,E1 -14322.076,E2 -14322.076} C_VEL
LIN {X 0,Y 345.22,Z 865.92,A -85,B 0,C 180,E1 -14323.831,E2 -14323.831} C_VEL
LIN {X 0,Y 346.198,Z 857.704,A -85,B 0,C 180,E1 -14325.293,E2 -14325.293} C_VEL
LIN {X 0,Y 347.253,Z 847.538,A -85,B 0,C 180,E1 -14326.753,E2 -14326.753} C_VEL
LIN {X 0,Y 348.349,Z 837.075,A -85,B 0,C 180,E1 -14327.948,E2 -14327.948} C_VEL
LIN {X 0,Y 349.247,Z 825.284,A -85,B 0,C 180,E1 -14329.02,E2 -14329.02} C_VEL
LIN {X 0,Y 349.913,Z 812.748,A -85,B 0,C 180,E1 -14329.871,E2 -14329.871} C_VEL
LIN {X 0,Y 350.246,Z 800.519,A -85,B 0,C 180,E1 -14330.471,E2 -14330.471} C_VEL
LIN {X 0,Y 350.349,Z 789.515,A -85,B 0,C 180,E1 -14330.827,E2 -14330.827} C_VEL
LIN {X 0,Y 349.729,Z 783.743,A -85,B 0,C 180,E1 -14331.009,E2 -14331.009} C_VEL
LIN {X 0,Y 344.535,Z 765.174,A -85,B 0,C 180,E1 -14331.763,E2 -14331.763} C_VEL
LIN {X 0,Y 344.041,Z 759.382,A -85,B 0,C 180,E1 -14331.922,E2 -14331.922} C_VEL
LIN {X 0,Y 344.441,Z 735.635,A -85,B 0,C 180,E1 -14332.422,E2 -14332.422} C_VEL
LIN {X 0,Y 334.871,Z 714.04,A -85,B 0,C 180,E1 -14333.63,E2 -14333.63} C_VEL
LIN {X 0,Y 333.74,Z 711.169,A -85,B 0,C 180,E1 -14333.786,E2 -14333.786} C_VEL
LIN {X 0,Y 333.695,Z 710.914,A -85,B 0,C 180,E1 -14333.907,E2 -14333.907} C_VEL
LIN {X 0,Y 333.714,Z 710.91,A -85,B 0,C 180,E1 -14337.59,E2 -14337.59} C_VEL
LIN {X 0,Y 333.662,Z 710.919,A -85,B 0,C 180,E1 -14340.354,E2 -14340.354} C_VEL
LIN {X 0,Y 333.641,Z 710.921,A -85,B 0,C 180,E1 -14344.65,E2 -14344.65} C_VEL
LIN {X 0,Y 333.618,Z 710.913,A -85,B 0,C 180,E1 -14347.642,E2 -14347.642} C_VEL
LIN {X 0,Y 333.66,Z 710.924,A -85,B 0,C 180,E1 -14350.751,E2 -14350.751} C_VEL
LIN {X 0,Y 333.686,Z 710.903,A -85,B 0,C 180,E1 -14354.266,E2 -14354.266} C_VEL
LIN {X 0,Y 333.659,Z 710.92,A -85,B 0,C 180,E1 -14357.621,E2 -14357.621} C_VEL
LIN {X 0,Y 333.629,Z 710.922,A -85,B 0,C 180,E1 -14361.189,E2 -14361.189} C_VEL
LIN {X 0,Y 333.631,Z 710.922,A -85,B 0,C 180,E1 -14365.22,E2 -14365.22} C_VEL
LIN {X 0,Y 333.588,Z 710.933,A -85,B 0,C 180,E1 -14368.217,E2 -14368.217} C_VEL
LIN {X 0,Y 333.652,Z 710.912,A -85,B 0,C 180,E1 -14371.022,E2 -14371.022} C_VEL
LIN {X 0,Y 333.674,Z 710.92,A -85,B 0,C 180,E1 -14373.748,E2 -14373.748} C_VEL
LIN {X 0,Y 333.657,Z 710.917,A -85,B 0,C 180,E1 -14377.91,E2 -14377.91} C_VEL
LIN {X 0,Y 333.728,Z 710.907,A -85,B 0,C 180,E1 -14381.586,E2 -14381.586} C_VEL
LIN {X 0,Y 333.742,Z 710.911,A -85,B 0,C 180,E1 -14385.574,E2 -14385.574} C_VEL
LIN {X 0,Y 333.769,Z 710.898,A -85,B 0,C 180,E1 -14389.076,E2 -14389.076} C_VEL
LIN {X 0,Y 333.945,Z 710.893,A -85,B 0,C 180,E1 -14392.746,E2 -14392.746} C_VEL
LIN {X 0,Y 333.751,Z 710.903,A -85,B 0,C 180,E1 -14395.168,E2 -14395.168} C_VEL
LIN {X 0,Y 334.07,Z 710.871,A -85,B 0,C 180,E1 -14397.588,E2 -14397.588} C_VEL
LIN {X 0,Y 334.197,Z 710.857,A -85,B 0,C 180,E1 -14400,E2 -14400} C_VEL
LIN {X 0,Y 334.07,Z 710.865,A -85,B 0,C 180,E1 -14402.411,E2 -14402.411} C_VEL
LIN {X 0,Y 333.945,Z 710.887,A -85,B 0,C 180,E1 -14407.254,E2 -14407.254} C_VEL
LIN {X 0,Y 333.769,Z 710.906,A -85,B 0,C 180,E1 -14410.924,E2 -14410.924} C_VEL
LIN {X 0,Y 333.742,Z 710.91,A -85,B 0,C 180,E1 -14414.637,E2 -14414.637} C_VEL
LIN {X 0,Y 333.73,Z 710.912,A -85,B 0,C 180,E1 -14418.658,E2 -14418.658} C_VEL
LIN {X 0,Y 333.598,Z 710.928,A -85,B 0,C 180,E1 -14422.285,E2 -14422.285} C_VEL
LIN {X 0,Y 333.675,Z 710.913,A -85,B 0,C 180,E1 -14426.251,E2 -14426.251} C_VEL
LIN {X 0,Y 333.653,Z 710.92,A -85,B 0,C 180,E1 -14428.978,E2 -14428.978} C_VEL
LIN {X 0,Y 333.595,Z 710.929,A -85,B 0,C 180,E1 -14432.595,E2 -14432.595} C_VEL
LIN {X 0,Y 333.624,Z 710.928,A -85,B 0,C 180,E1 -14436.146,E2 -14436.146} C_VEL
LIN {X 0,Y 333.633,Z 710.908,A -85,B 0,C 180,E1 -14439.194,E2 -14439.194} C_VEL
LIN {X 0,Y 333.656,Z 710.922,A -85,B 0,C 180,E1 -14442.521,E2 -14442.521} C_VEL
LIN {X 0,Y 333.686,Z 710.921,A -85,B 0,C 180,E1 -14445.985,E2 -14445.985} C_VEL
LIN {X 0,Y 333.662,Z 710.924,A -85,B 0,C 180,E1 -14449.313,E2 -14449.313} C_VEL
LIN {X 0,Y 333.68,Z 711.103,A -85,B 0,C 180,E1 -14452.636,E2 -14452.636} C_VEL
LIN {X 0,Y 337.048,Z 724.209,A -85,B 0,C 180,E1 -14455.749,E2 -14455.749} C_VEL
LIN {X 0,Y 340.522,Z 740.124,A -85,B 0,C 180,E1 -14459.271,E2 -14459.271} C_VEL
LIN {X 0,Y 340.686,Z 743.35,A -85,B 0,C 180,E1 -14459.927,E2 -14459.927} C_VEL
LIN {X 0,Y 338.068,Z 765.355,A -85,B 0,C 180,E1 -14464.126,E2 -14464.126} C_VEL
LIN {X 0,Y 337.08,Z 774.856,A -85,B 0,C 180,E1 -14465.956,E2 -14465.956} C_VEL
LIN {X 0,Y 341.224,Z 810.283,A -85,B 0,C 180,E1 -14467.053,E2 -14467.053} C_VEL
LIN {X 0,Y 343.091,Z 830.995,A -85,B 0,C 180,E1 -14467.636,E2 -14467.636} C_VEL
LIN {X 0,Y 341.805,Z 886.216,A -85,B 0,C 180,E1 -14468.802,E2 -14468.802} C_VEL
LIN {X 0,Y 341.071,Z 900.161,A -85,B 0,C 180,E1 -14469.347,E2 -14469.347} C_VEL
LIN {X 0,Y 339.939,Z 912.658,A -85,B 0,C 180,E1 -14470.064,E2 -14470.064} C_VEL
LIN {X 0,Y 338.701,Z 923.844,A -85,B 0,C 180,E1 -14470.934,E2 -14470.934} C_VEL
LIN {X 0,Y 337.203,Z 935.51,A -85,B 0,C 180,E1 -14472.106,E2 -14472.106} C_VEL
LIN {X 0,Y 335.862,Z 946.063,A -85,B 0,C 180,E1 -14473.444,E2 -14473.444} C_VEL
LIN {X 0,Y 334.881,Z 954.674,A -85,B 0,C 180,E1 -14474.789,E2 -14474.789} C_VEL
LIN {X 0,Y 334.085,Z 962.797,A -85,B 0,C 180,E1 -14476.32,E2 -14476.32} C_VEL
LIN {X 0,Y 333.267,Z 970.68,A -85,B 0,C 180,E1 -14478.144,E2 -14478.144} C_VEL
LIN {X 0,Y 332.781,Z 978,A -85,B 0,C 180,E1 -14480.282,E2 -14480.282} C_VEL
LIN {X 0,Y 332.685,Z 982.912,A -85,B 0,C 180,E1 -14482.116,E2 -14482.116} C_VEL
LIN {X 0,Y 332.781,Z 986.697,A -85,B 0,C 180,E1 -14483.947,E2 -14483.947} C_VEL
LIN {X 0,Y 332.937,Z 988.663,A -85,B 0,C 180,E1 -14485.165,E2 -14485.165} C_VEL
LIN {X 0,Y 333.052,Z 990.136,A -85,B 0,C 180,E1 -14486.379,E2 -14486.379} C_VEL
LIN {X 0,Y 333.102,Z 991.181,A -85,B 0,C 180,E1 -14487.59,E2 -14487.59} C_VEL
LIN {X 0,Y 333.189,Z 991.825,A -85,B 0,C 180,E1 -14488.799,E2 -14488.799} C_VEL
LIN {X 0,Y 333.267,Z 992.056,A -85,B 0,C 180,E1 -14490.008,E2 -14490.008} C_VEL
LIN {X 0,Y 333.189,Z 991.813,A -85,B 0,C 180,E1 -14491.217,E2 -14491.217} C_VEL
LIN {X 0,Y 333.104,Z 991.161,A -85,B 0,C 180,E1 -14492.426,E2 -14492.426} C_VEL
LIN {X 0,Y 333.054,Z 990.107,A -85,B 0,C 180,E1 -14493.637,E2 -14493.637} C_VEL
LIN {X 0,Y 332.934,Z 988.621,A -85,B 0,C 180,E1 -14494.851,E2 -14494.851} C_VEL
LIN {X 0,Y 332.724,Z 985.069,A -85,B 0,C 180,E1 -14496.896,E2 -14496.896} C_VEL
LIN {X 0,Y 332.737,Z 979.688,A -85,B 0,C 180,E1 -14499.122,E2 -14499.122} C_VEL
LIN {X 0,Y 332.966,Z 973.937,A -85,B 0,C 180,E1 -14500.958,E2 -14500.958} C_VEL
LIN {X 0,Y 333.593,Z 966.826,A -85,B 0,C 180,E1 -14502.787,E2 -14502.787} C_VEL
LIN {X 0,Y 334.285,Z 959.588,A -85,B 0,C 180,E1 -14504.309,E2 -14504.309} C_VEL
LIN {X 0,Y 335.424,Z 950.928,A -85,B 0,C 180,E1 -14505.813,E2 -14505.813} C_VEL
LIN {X 0,Y 336.485,Z 941.417,A -85,B 0,C 180,E1 -14507.166,E2 -14507.166} C_VEL
LIN {X 0,Y 337.971,Z 930.655,A -85,B 0,C 180,E1 -14508.496,E2 -14508.496} C_VEL
LIN {X 0,Y 339.62,Z 919.297,A -85,B 0,C 180,E1 -14509.657,E2 -14509.657} C_VEL
LIN {X 0,Y 341.481,Z 904.983,A -85,B 0,C 180,E1 -14510.802,E2 -14510.802} C_VEL
LIN {X 0,Y 342.938,Z 892.412,A -85,B 0,C 180,E1 -14511.535,E2 -14511.535} C_VEL
LIN {X 0,Y 343.905,Z 881.421,A -85,B 0,C 180,E1 -14512.023,E2 -14512.023} C_VEL
LIN {X 0,Y 346.757,Z 829.542,A -85,B 0,C 180,E1 -14513.718,E2 -14513.718} C_VEL
LIN {X 0,Y 345.6,Z 802.664,A -85,B 0,C 180,E1 -14514.956,E2 -14514.956} C_VEL
LIN {X 0,Y 343.643,Z 783.798,A -85,B 0,C 180,E1 -14516.037,E2 -14516.037} C_VEL
LIN {X 0,Y 341.228,Z 765.763,A -85,B 0,C 180,E1 -14517.227,E2 -14517.227} C_VEL
LIN {X 0,Y 339.415,Z 753.399,A -85,B 0,C 180,E1 -14518.144,E2 -14518.144} C_VEL
LIN {X 0,Y 340.656,Z 743.32,A -85,B 0,C 180,E1 -14520.064,E2 -14520.064} C_VEL
LIN {X 0,Y 340.412,Z 739.975,A -85,B 0,C 180,E1 -14520.748,E2 -14520.748} C_VEL
LIN {X 0,Y 337.615,Z 726.865,A -85,B 0,C 180,E1 -14523.626,E2 -14523.626} C_VEL
LIN {X 0,Y 334.119,Z 712.756,A -85,B 0,C 180,E1 -14526.936,E2 -14526.936} C_VEL
LIN {X 0,Y 333.694,Z 710.917,A -85,B 0,C 180,E1 -14527.423,E2 -14527.423} C_VEL
LIN {X 0,Y 333.616,Z 710.926,A -85,B 0,C 180,E1 -14530.779,E2 -14530.779} C_VEL
LIN {X 0,Y 333.601,Z 710.927,A -85,B 0,C 180,E1 -14534.252,E2 -14534.252} C_VEL
LIN {X 0,Y 333.64,Z 710.927,A -85,B 0,C 180,E1 -14537.618,E2 -14537.618} C_VEL
LIN {X 0,Y 333.637,Z 710.925,A -85,B 0,C 180,E1 -14541.213,E2 -14541.213} C_VEL
LIN {X 0,Y 333.694,Z 710.919,A -85,B 0,C 180,E1 -14543.863,E2 -14543.863} C_VEL
LIN {X 0,Y 333.662,Z 710.925,A -85,B 0,C 180,E1 -14547.417,E2 -14547.417} C_VEL
LIN {X 0,Y 333.673,Z 710.924,A -85,B 0,C 180,E1 -14551.024,E2 -14551.024} C_VEL
LIN {X 0,Y 334.665,Z 713.774,A -85,B 0,C 180,E1 -14551.442,E2 -14551.442} C_VEL
LIN {X 0,Y 336.939,Z 716.341,A -85,B 0,C 180,E1 -14552.084,E2 -14552.084} C_VEL
LIN {X 0,Y 338.992,Z 719.708,A -85,B 0,C 180,E1 -14552.672,E2 -14552.672} C_VEL
LIN {X 0,Y 340.207,Z 721.487,A -85,B 0,C 180,E1 -14553.003,E2 -14553.003} C_VEL
LIN {X 0,Y 343.18,Z 726.313,A -85,B 0,C 180,E1 -14553.795,E2 -14553.795} C_VEL
LIN {X 0,Y 347.746,Z 734.211,A -85,B 0,C 180,E1 -14554.934,E2 -14554.934} C_VEL
LIN {X 0,Y 351.397,Z 741.567,A -85,B 0,C 180,E1 -14555.797,E2 -14555.797} C_VEL
LIN {X 0,Y 348.301,Z 788.609,A -85,B 0,C 180,E1 -14557.367,E2 -14557.367} C_VEL
LIN {X 0,Y 347.851,Z 804.396,A -85,B 0,C 180,E1 -14557.985,E2 -14557.985} C_VEL
LIN {X 0,Y 347.368,Z 815.143,A -85,B 0,C 180,E1 -14558.552,E2 -14558.552} C_VEL
LIN {X 0,Y 346.66,Z 825.489,A -85,B 0,C 180,E1 -14559.257,E2 -14559.257} C_VEL
LIN {X 0,Y 345.773,Z 835.478,A -85,B 0,C 180,E1 -14560.096,E2 -14560.096} C_VEL
LIN {X 0,Y 344.935,Z 843.986,A -85,B 0,C 180,E1 -14560.974,E2 -14560.974} C_VEL
LIN {X 0,Y 343.959,Z 851.285,A -85,B 0,C 180,E1 -14561.844,E2 -14561.844} C_VEL
LIN {X 0,Y 342.876,Z 859.437,A -85,B 0,C 180,E1 -14563.017,E2 -14563.017} C_VEL
LIN {X 0,Y 341.776,Z 866.352,A -85,B 0,C 180,E1 -14564.189,E2 -14564.189} C_VEL
LIN {X 0,Y 340.74,Z 872.332,A -85,B 0,C 180,E1 -14565.365,E2 -14565.365} C_VEL
LIN {X 0,Y 339.605,Z 878.548,A -85,B 0,C 180,E1 -14566.842,E2 -14566.842} C_VEL
LIN {X 0,Y 338.757,Z 882.794,A -85,B 0,C 180,E1 -14568.026,E2 -14568.026} C_VEL
LIN {X 0,Y 337.634,Z 887.867,A -85,B 0,C 180,E1 -14569.809,E2 -14569.809} C_VEL
LIN {X 0,Y 336.518,Z 891.753,A -85,B 0,C 180,E1 -14571.594,E2 -14571.594} C_VEL
LIN {X 0,Y 335.899,Z 893.761,A -85,B 0,C 180,E1 -14572.788,E2 -14572.788} C_VEL
LIN {X 0,Y 335.142,Z 896.238,A -85,B 0,C 180,E1 -14575.188,E2 -14575.188} C_VEL
LIN {X 0,Y 334.83,Z 896.871,A -85,B 0,C 180,E1 -14576.39,E2 -14576.39} C_VEL
LIN {X 0,Y 334.502,Z 897.053,A -85,B 0,C 180,E1 -14577.592,E2 -14577.592} C_VEL
LIN {X 0,Y 334.293,Z 896.756,A -85,B 0,C 180,E1 -14578.795,E2 -14578.795} C_VEL
LIN {X 0,Y 333.985,Z 896.073,A -85,B 0,C 180,E1 -14580,E2 -14580} C_VEL
LIN {X 0,Y 333.82,Z 893.28,A -85,B 0,C 180,E1 -14582.413,E2 -14582.413} C_VEL
LIN {X 0,Y 333.654,Z 891.301,A -85,B 0,C 180,E1 -14583.623,E2 -14583.623} C_VEL
LIN {X 0,Y 334.03,Z 887.294,A -85,B 0,C 180,E1 -14585.433,E2 -14585.433} C_VEL
LIN {X 0,Y 334.388,Z 881.057,A -85,B 0,C 180,E1 -14587.548,E2 -14587.548} C_VEL
LIN {X 0,Y 334.724,Z 874.613,A -85,B 0,C 180,E1 -14589.284,E2 -14589.284} C_VEL
LIN {X 0,Y 335.054,Z 868.902,A -85,B 0,C 180,E1 -14590.576,E2 -14590.576} C_VEL
LIN {X 0,Y 335.58,Z 860.924,A -85,B 0,C 180,E1 -14592.089,E2 -14592.089} C_VEL
LIN {X 0,Y 336.067,Z 852.33,A -85,B 0,C 180,E1 -14593.453,E2 -14593.453} C_VEL
LIN {X 0,Y 336.502,Z 844.459,A -85,B 0,C 180,E1 -14594.515,E2 -14594.515} C_VEL
LIN {X 0,Y 337.09,Z 835.171,A -85,B 0,C 180,E1 -14595.571,E2 -14595.571} C_VEL
LIN {X 0,Y 337.551,Z 825.723,A -85,B 0,C 180,E1 -14596.47,E2 -14596.47} C_VEL
LIN {X 0,Y 337.946,Z 815.92,A -85,B 0,C 180,E1 -14597.238,E2 -14597.238} C_VEL
LIN {X 0,Y 338.282,Z 804.935,A -85,B 0,C 180,E1 -14597.923,E2 -14597.923} C_VEL
LIN {X 0,Y 338.506,Z 794.479,A -85,B 0,C 180,E1 -14598.419,E2 -14598.419} C_VEL
LIN {X 0,Y 338.659,Z 780.597,A -85,B 0,C 180,E1 -14598.881,E2 -14598.881} C_VEL
LIN {X 0,Y 339.786,Z 729.899,A -85,B 0,C 180,E1 -14600.291,E2 -14600.291} C_VEL
LIN {X 0,Y 333.752,Z 710.91,A -85,B 0,C 180,E1 -14601.117,E2 -14601.117} C_VEL
LIN {X 0,Y 333.711,Z 710.916,A -85,B 0,C 180,E1 -14605.087,E2 -14605.087} C_VEL
LIN {X 0,Y 333.673,Z 710.924,A -85,B 0,C 180,E1 -14608.976,E2 -14608.976} C_VEL
LIN {X 0,Y 333.662,Z 710.923,A -85,B 0,C 180,E1 -14612.583,E2 -14612.583} C_VEL
LIN {X 0,Y 333.694,Z 710.914,A -85,B 0,C 180,E1 -14616.137,E2 -14616.137} C_VEL
LIN {X 0,Y 333.623,Z 710.925,A -85,B 0,C 180,E1 -14619.196,E2 -14619.196} C_VEL
LIN {X 0,Y 333.647,Z 710.919,A -85,B 0,C 180,E1 -14622.495,E2 -14622.495} C_VEL
LIN {X 0,Y 333.613,Z 710.922,A -85,B 0,C 180,E1 -14625.951,E2 -14625.951} C_VEL
LIN {X 0,Y 333.622,Z 710.923,A -85,B 0,C 180,E1 -14629.321,E2 -14629.321} C_VEL
LIN {X 0,Y 333.68,Z 710.915,A -85,B 0,C 180,E1 -14633.165,E2 -14633.165} C_VEL
LIN {X 0,Y 333.692,Z 710.914,A -85,B 0,C 180,E1 -14635.336,E2 -14635.336} C_VEL
LIN {X 0,Y 333.638,Z 710.92,A -85,B 0,C 180,E1 -14638.216,E2 -14638.216} C_VEL
LIN {X 0,Y 333.641,Z 710.921,A -85,B 0,C 180,E1 -14641.014,E2 -14641.014} C_VEL
LIN {X 0,Y 333.671,Z 710.921,A -85,B 0,C 180,E1 -14644.917,E2 -14644.917} C_VEL
LIN {X 0,Y 333.683,Z 710.919,A -85,B 0,C 180,E1 -14646.311,E2 -14646.311} C_VEL
LIN {X 0,Y 334.769,Z 713.849,A -85,B 0,C 180,E1 -14646.469,E2 -14646.469} C_VEL
LIN {X 0,Y 343.735,Z 733.987,A -85,B 0,C 180,E1 -14647.6,E2 -14647.6} C_VEL
LIN {X 0,Y 344.457,Z 736.289,A -85,B 0,C 180,E1 -14647.703,E2 -14647.703} C_VEL
LIN {X 0,Y 343.668,Z 787.054,A -85,B 0,C 180,E1 -14648.774,E2 -14648.774} C_VEL
LIN {X 0,Y 343.634,Z 799.952,A -85,B 0,C 180,E1 -14649.158,E2 -14649.158} C_VEL
LIN {X 0,Y 343.279,Z 812.85,A -85,B 0,C 180,E1 -14649.782,E2 -14649.782} C_VEL
LIN {X 0,Y 342.627,Z 824.387,A -85,B 0,C 180,E1 -14650.554,E2 -14650.554} C_VEL
LIN {X 0,Y 341.767,Z 835.974,A -85,B 0,C 180,E1 -14651.572,E2 -14651.572} C_VEL
LIN {X 0,Y 340.731,Z 846.448,A -85,B 0,C 180,E1 -14652.745,E2 -14652.745} C_VEL
LIN {X 0,Y 339.639,Z 856.049,A -85,B 0,C 180,E1 -14654.08,E2 -14654.08} C_VEL
LIN {X 0,Y 338.672,Z 864.746,A -85,B 0,C 180,E1 -14655.573,E2 -14655.573} C_VEL
LIN {X 0,Y 337.421,Z 873.252,A -85,B 0,C 180,E1 -14657.36,E2 -14657.36} C_VEL
LIN {X 0,Y 336.375,Z 880.016,A -85,B 0,C 180,E1 -14659.154,E2 -14659.154} C_VEL
LIN {X 0,Y 335.803,Z 885.383,A -85,B 0,C 180,E1 -14660.962,E2 -14660.962} C_VEL
LIN {X 0,Y 335.408,Z 888.32,A -85,B 0,C 180,E1 -14662.165,E2 -14662.165} C_VEL
LIN {X 0,Y 334.597,Z 891.881,A -85,B 0,C 180,E1 -14663.964,E2 -14663.964} C_VEL
LIN {X 0,Y 334.295,Z 893.705,A -85,B 0,C 180,E1 -14665.168,E2 -14665.168} C_VEL
LIN {X 0,Y 334.186,Z 895.062,A -85,B 0,C 180,E1 -14666.375,E2 -14666.375} C_VEL
LIN {X 0,Y 334.157,Z 896.019,A -85,B 0,C 180,E1 -14667.581,E2 -14667.581} C_VEL
LIN {X 0,Y 333.964,Z 896.862,A -85,B 0,C 180,E1 -14669.992,E2 -14669.992} C_VEL
LIN {X 0,Y 334.161,Z 896.099,A -85,B 0,C 180,E1 -14672.403,E2 -14672.403} C_VEL
LIN {X 0,Y 334.278,Z 893.869,A -85,B 0,C 180,E1 -14674.816,E2 -14674.816} C_VEL
LIN {X 0,Y 334.794,Z 891.055,A -85,B 0,C 180,E1 -14676.621,E2 -14676.621} C_VEL
LIN {X 0,Y 335.528,Z 887.229,A -85,B 0,C 180,E1 -14678.423,E2 -14678.423} C_VEL
LIN {X 0,Y 336.218,Z 881.758,A -85,B 0,C 180,E1 -14680.415,E2 -14680.415} C_VEL
LIN {X 0,Y 337.206,Z 874.947,A -85,B 0,C 180,E1 -14682.326,E2 -14682.326} C_VEL
LIN {X 0,Y 338.401,Z 866.92,A -85,B 0,C 180,E1 -14684.115,E2 -14684.115} C_VEL
LIN {X 0,Y 339.424,Z 858.704,A -85,B 0,C 180,E1 -14685.606,E2 -14685.606} C_VEL
LIN {X 0,Y 340.529,Z 848.537,A -85,B 0,C 180,E1 -14687.094,E2 -14687.094} C_VEL
LIN {X 0,Y 341.665,Z 838.068,A -85,B 0,C 180,E1 -14688.312,E2 -14688.312} C_VEL
LIN {X 0,Y 342.609,Z 826.281,A -85,B 0,C 180,E1 -14689.403,E2 -14689.403} C_VEL
LIN {X 0,Y 343.328,Z 813.739,A -85,B 0,C 180,E1 -14690.269,E2 -14690.269} C_VEL
LIN {X 0,Y 343.653,Z 801.693,A -85,B 0,C 180,E1 -14690.875,E2 -14690.875} C_VEL
LIN {X 0,Y 343.789,Z 790.041,A -85,B 0,C 180,E1 -14691.255,E2 -14691.255} C_VEL
LIN {X 0,Y 344.041,Z 759.382,A -85,B 0,C 180,E1 -14691.922,E2 -14691.922} C_VEL
LIN {X 0,Y 343.673,Z 753.502,A -85,B 0,C 180,E1 -14692.079,E2 -14692.079} C_VEL
LIN {X 0,Y 342.443,Z 747.79,A -85,B 0,C 180,E1 -14692.294,E2 -14692.294} C_VEL
LIN {X 0,Y 339.83,Z 740.48,A -85,B 0,C 180,E1 -14692.649,E2 -14692.649} C_VEL
LIN {X 0,Y 334.729,Z 730.063,A -85,B 0,C 180,E1 -14693.272,E2 -14693.272} C_VEL
LIN {X 0,Y 326.819,Z 712.6,A -85,B 0,C 180,E1 -14694.313,E2 -14694.313} C_VEL
LIN {X 0,Y 326.68,Z 711.787,A -85,B 0,C 180,E1 -14694.37,E2 -14694.37} C_VEL
LIN {X 0,Y 326.624,Z 711.793,A -85,B 0,C 180,E1 -14698.242,E2 -14698.242} C_VEL
LIN {X 0,Y 326.561,Z 711.808,A -85,B 0,C 180,E1 -14701.086,E2 -14701.086} C_VEL
LIN {X 0,Y 326.575,Z 711.802,A -85,B 0,C 180,E1 -14704.011,E2 -14704.011} C_VEL
LIN {X 0,Y 326.593,Z 711.793,A -85,B 0,C 180,E1 -14707.23,E2 -14707.23} C_VEL
LIN {X 0,Y 326.596,Z 711.804,A -85,B 0,C 180,E1 -14710.194,E2 -14710.194} C_VEL
LIN {X 0,Y 326.616,Z 711.791,A -85,B 0,C 180,E1 -14713.502,E2 -14713.502} C_VEL
LIN {X 0,Y 326.604,Z 711.794,A -85,B 0,C 180,E1 -14717.007,E2 -14717.007} C_VEL
LIN {X 0,Y 326.594,Z 711.798,A -85,B 0,C 180,E1 -14720.759,E2 -14720.759} C_VEL
LIN {X 0,Y 326.559,Z 711.804,A -85,B 0,C 180,E1 -14724.473,E2 -14724.473} C_VEL
LIN {X 0,Y 326.559,Z 711.803,A -85,B 0,C 180,E1 -14727.45,E2 -14727.45} C_VEL
LIN {X 0,Y 326.604,Z 711.792,A -85,B 0,C 180,E1 -14730.335,E2 -14730.335} C_VEL
LIN {X 0,Y 326.629,Z 711.796,A -85,B 0,C 180,E1 -14734.511,E2 -14734.511} C_VEL
LIN {X 0,Y 326.582,Z 711.805,A -85,B 0,C 180,E1 -14738.541,E2 -14738.541} C_VEL
LIN {X 0,Y 326.681,Z 711.785,A -85,B 0,C 180,E1 -14741.174,E2 -14741.174} C_VEL
LIN {X 0,Y 326.697,Z 711.789,A -85,B 0,C 180,E1 -14745.43,E2 -14745.43} C_VEL
LIN {X 0,Y 326.705,Z 711.778,A -85,B 0,C 180,E1 -14748.837,E2 -14748.837} C_VEL
LIN {X 0,Y 326.899,Z 711.769,A -85,B 0,C 180,E1 -14752.588,E2 -14752.588} C_VEL
LIN {X 0,Y 326.717,Z 711.78,A -85,B 0,C 180,E1 -14755.064,E2 -14755.064} C_VEL
LIN {X 0,Y 327.007,Z 711.751,A -85,B 0,C 180,E1 -14757.536,E2 -14757.536} C_VEL
LIN {X 0,Y 327.148,Z 711.735,A -85,B 0,C 180,E1 -14760,E2 -14760} C_VEL
LIN {X 0,Y 327.008,Z 711.744,A -85,B 0,C 180,E1 -14762.463,E2 -14762.463} C_VEL
LIN {X 0,Y 326.924,Z 711.763,A -85,B 0,C 180,E1 -14766.17,E2 -14766.17} C_VEL
LIN {X 0,Y 326.746,Z 711.778,A -85,B 0,C 180,E1 -14769.908,E2 -14769.908} C_VEL
LIN {X 0,Y 326.69,Z 711.791,A -85,B 0,C 180,E1 -14773.688,E2 -14773.688} C_VEL
LIN {X 0,Y 326.633,Z 711.799,A -85,B 0,C 180,E1 -14777.532,E2 -14777.532} C_VEL
LIN {X 0,Y 326.593,Z 711.792,A -85,B 0,C 180,E1 -14780.14,E2 -14780.14} C_VEL
LIN {X 0,Y 326.589,Z 711.8,A -85,B 0,C 180,E1 -14784.134,E2 -14784.134} C_VEL
LIN {X 0,Y 326.625,Z 711.792,A -85,B 0,C 180,E1 -14786.863,E2 -14786.863} C_VEL
LIN {X 0,Y 326.585,Z 711.797,A -85,B 0,C 180,E1 -14790.618,E2 -14790.618} C_VEL
LIN {X 0,Y 326.554,Z 711.803,A -85,B 0,C 180,E1 -14794.026,E2 -14794.026} C_VEL
LIN {X 0,Y 326.578,Z 711.801,A -85,B 0,C 180,E1 -14797.246,E2 -14797.246} C_VEL
LIN {X 0,Y 326.586,Z 711.794,A -85,B 0,C 180,E1 -14800.21,E2 -14800.21} C_VEL
LIN {X 0,Y 326.612,Z 711.8,A -85,B 0,C 180,E1 -14803.517,E2 -14803.517} C_VEL
LIN {X 0,Y 326.608,Z 711.794,A -85,B 0,C 180,E1 -14807.022,E2 -14807.022} C_VEL
LIN {X 0,Y 326.606,Z 711.796,A -85,B 0,C 180,E1 -14810.774,E2 -14810.774} C_VEL
LIN {X 0,Y 326.63,Z 711.956,A -85,B 0,C 180,E1 -14812.118,E2 -14812.118} C_VEL
LIN {X 0,Y 329.937,Z 724.824,A -85,B 0,C 180,E1 -14815.265,E2 -14815.265} C_VEL
LIN {X 0,Y 333.108,Z 739.129,A -85,B 0,C 180,E1 -14818.533,E2 -14818.533} C_VEL
LIN {X 0,Y 333.81,Z 742.664,A -85,B 0,C 180,E1 -14819.311,E2 -14819.311} C_VEL
LIN {X 0,Y 333.402,Z 747.73,A -85,B 0,C 180,E1 -14820.317,E2 -14820.317} C_VEL
LIN {X 0,Y 330.832,Z 769.253,A -85,B 0,C 180,E1 -14824.532,E2 -14824.532} C_VEL
LIN {X 0,Y 330.287,Z 773.854,A -85,B 0,C 180,E1 -14825.438,E2 -14825.438} C_VEL
LIN {X 0,Y 334.558,Z 809.938,A -85,B 0,C 180,E1 -14826.584,E2 -14826.584} C_VEL
LIN {X 0,Y 336.5,Z 831.484,A -85,B 0,C 180,E1 -14827.207,E2 -14827.207} C_VEL
LIN {X 0,Y 335.226,Z 885.221,A -85,B 0,C 180,E1 -14828.365,E2 -14828.365} C_VEL
LIN {X 0,Y 334.469,Z 898.388,A -85,B 0,C 180,E1 -14828.88,E2 -14828.88} C_VEL
LIN {X 0,Y 333.254,Z 911.649,A -85,B 0,C 180,E1 -14829.647,E2 -14829.647} C_VEL
LIN {X 0,Y 331.789,Z 924.429,A -85,B 0,C 180,E1 -14830.682,E2 -14830.682} C_VEL
LIN {X 0,Y 330.242,Z 935.801,A -85,B 0,C 180,E1 -14831.876,E2 -14831.876} C_VEL
LIN {X 0,Y 328.877,Z 946.103,A -85,B 0,C 180,E1 -14833.242,E2 -14833.242} C_VEL
LIN {X 0,Y 327.943,Z 954.089,A -85,B 0,C 180,E1 -14834.535,E2 -14834.535} C_VEL
LIN {X 0,Y 326.924,Z 963.182,A -85,B 0,C 180,E1 -14836.331,E2 -14836.331} C_VEL
LIN {X 0,Y 326.146,Z 970.812,A -85,B 0,C 180,E1 -14838.197,E2 -14838.197} C_VEL
LIN {X 0,Y 325.74,Z 976.982,A -85,B 0,C 180,E1 -14840.07,E2 -14840.07} C_VEL
LIN {X 0,Y 325.604,Z 981.893,A -85,B 0,C 180,E1 -14841.944,E2 -14841.944} C_VEL
LIN {X 0,Y 325.72,Z 985.684,A -85,B 0,C 180,E1 -14843.815,E2 -14843.815} C_VEL
LIN {X 0,Y 325.883,Z 987.653,A -85,B 0,C 180,E1 -14845.06,E2 -14845.06} C_VEL
LIN {X 0,Y 326.008,Z 989.129,A -85,B 0,C 180,E1 -14846.3,E2 -14846.3} C_VEL
LIN {X 0,Y 326.058,Z 990.176,A -85,B 0,C 180,E1 -14847.538,E2 -14847.538} C_VEL
LIN {X 0,Y 326.152,Z 990.821,A -85,B 0,C 180,E1 -14848.774,E2 -14848.774} C_VEL
LIN {X 0,Y 326.237,Z 991.053,A -85,B 0,C 180,E1 -14850.008,E2 -14850.008} C_VEL
LIN {X 0,Y 326.152,Z 990.809,A -85,B 0,C 180,E1 -14851.243,E2 -14851.243} C_VEL
LIN {X 0,Y 326.06,Z 990.155,A -85,B 0,C 180,E1 -14852.479,E2 -14852.479} C_VEL
LIN {X 0,Y 326.01,Z 989.099,A -85,B 0,C 180,E1 -14853.716,E2 -14853.716} C_VEL
LIN {X 0,Y 325.858,Z 987.607,A -85,B 0,C 180,E1 -14854.957,E2 -14854.957} C_VEL
LIN {X 0,Y 325.671,Z 984.288,A -85,B 0,C 180,E1 -14856.933,E2 -14856.933} C_VEL
LIN {X 0,Y 325.632,Z 980.331,A -85,B 0,C 180,E1 -14858.697,E2 -14858.697} C_VEL
LIN {X 0,Y 325.869,Z 973.96,A -85,B 0,C 180,E1 -14860.885,E2 -14860.885} C_VEL
LIN {X 0,Y 326.483,Z 967.072,A -85,B 0,C 180,E1 -14862.754,E2 -14862.754} C_VEL
LIN {X 0,Y 327.212,Z 960.134,A -85,B 0,C 180,E1 -14864.299,E2 -14864.299} C_VEL
LIN {X 0,Y 327.78,Z 955.291,A -85,B 0,C 180,E1 -14865.234,E2 -14865.234} C_VEL
LIN {X 0,Y 329.512,Z 942.445,A -85,B 0,C 180,E1 -14867.381,E2 -14867.381} C_VEL
LIN {X 0,Y 331.093,Z 932.399,A -85,B 0,C 180,E1 -14868.734,E2 -14868.734} C_VEL
LIN {X 0,Y 332.734,Z 921.666,A -85,B 0,C 180,E1 -14869.92,E2 -14869.92} C_VEL
LIN {X 0,Y 334.205,Z 912.017,A -85,B 0,C 180,E1 -14870.792,E2 -14870.792} C_VEL
LIN {X 0,Y 335.636,Z 901.404,A -85,B 0,C 180,E1 -14871.584,E2 -14871.584} C_VEL
LIN {X 0,Y 337.008,Z 889.91,A -85,B 0,C 180,E1 -14872.256,E2 -14872.256} C_VEL
LIN {X 0,Y 338.023,Z 878.837,A -85,B 0,C 180,E1 -14872.749,E2 -14872.749} C_VEL
LIN {X 0,Y 340.95,Z 830.4,A -85,B 0,C 180,E1 -14874.38,E2 -14874.38} C_VEL
LIN {X 0,Y 339.96,Z 803.775,A -85,B 0,C 180,E1 -14875.657,E2 -14875.657} C_VEL
LIN {X 0,Y 338.303,Z 786.224,A -85,B 0,C 180,E1 -14876.709,E2 -14876.709} C_VEL
LIN {X 0,Y 336.191,Z 768.758,A -85,B 0,C 180,E1 -14877.908,E2 -14877.908} C_VEL
LIN {X 0,Y 334.079,Z 754.757,A -85,B 0,C 180,E1 -14879.004,E2 -14879.004} C_VEL
LIN {X 0,Y 333.336,Z 748.761,A -85,B 0,C 180,E1 -14879.534,E2 -14879.534} C_VEL
LIN {X 0,Y 333.546,Z 746.427,A -85,B 0,C 180,E1 -14879.922,E2 -14879.922} C_VEL
LIN {X 0,Y 333.691,Z 742.468,A -85,B 0,C 180,E1 -14880.72,E2 -14880.72} C_VEL
LIN {X 0,Y 331.124,Z 730.036,A -85,B 0,C 180,E1 -14883.5,E2 -14883.5} C_VEL
LIN {X 0,Y 328.081,Z 717.526,A -85,B 0,C 180,E1 -14886.476,E2 -14886.476} C_VEL
LIN {X 0,Y 326.618,Z 711.801,A -85,B 0,C 180,E1 -14887.898,E2 -14887.898} C_VEL
LIN {X 0,Y 326.567,Z 711.806,A -85,B 0,C 180,E1 -14891.855,E2 -14891.855} C_VEL
LIN {X 0,Y 326.539,Z 711.81,A -85,B 0,C 180,E1 -14895.263,E2 -14895.263} C_VEL
LIN {X 0,Y 326.556,Z 711.805,A -85,B 0,C 180,E1 -14898.881,E2 -14898.881} C_VEL
LIN {X 0,Y 326.642,Z 711.794,A -85,B 0,C 180,E1 -14902.766,E2 -14902.766} C_VEL
LIN {X 0,Y 326.627,Z 711.798,A -85,B 0,C 180,E1 -14905.983,E2 -14905.983} C_VEL
LIN {X 0,Y 326.612,Z 711.803,A -85,B 0,C 180,E1 -14909.364,E2 -14909.364} C_VEL
LIN {X 0,Y 327.6,Z 714.593,A -85,B 0,C 180,E1 -14909.819,E2 -14909.819} C_VEL
LIN {X 0,Y 329.725,Z 716.815,A -85,B 0,C 180,E1 -14910.509,E2 -14910.509} C_VEL
LIN {X 0,Y 332.253,Z 720.834,A -85,B 0,C 180,E1 -14911.343,E2 -14911.343} C_VEL
LIN {X 0,Y 333.388,Z 722.189,A -85,B 0,C 180,E1 -14911.677,E2 -14911.677} C_VEL
LIN {X 0,Y 338.608,Z 730.532,A -85,B 0,C 180,E1 -14913.197,E2 -14913.197} C_VEL
LIN {X 0,Y 343.371,Z 739.018,A -85,B 0,C 180,E1 -14914.458,E2 -14914.458} C_VEL
LIN {X 0,Y 345.841,Z 744.373,A -85,B 0,C 180,E1 -14915.119,E2 -14915.119} C_VEL
LIN {X 0,Y 342.564,Z 791.296,A -85,B 0,C 180,E1 -14916.738,E2 -14916.738} C_VEL
LIN {X 0,Y 341.999,Z 807.414,A -85,B 0,C 180,E1 -14917.417,E2 -14917.417} C_VEL
LIN {X 0,Y 341.455,Z 817.796,A -85,B 0,C 180,E1 -14917.993,E2 -14917.993} C_VEL
LIN {X 0,Y 340.658,Z 828.385,A -85,B 0,C 180,E1 -14918.748,E2 -14918.748} C_VEL
LIN {X 0,Y 339.605,Z 839.184,A -85,B 0,C 180,E1 -14919.718,E2 -14919.718} C_VEL
LIN {X 0,Y 338.083,Z 850.906,A -85,B 0,C 180,E1 -14921.046,E2 -14921.046} C_VEL
LIN {X 0,Y 336.789,Z 860.235,A -85,B 0,C 180,E1 -14922.387,E2 -14922.387} C_VEL
LIN {X 0,Y 335.607,Z 867.254,A -85,B 0,C 180,E1 -14923.578,E2 -14923.578} C_VEL
LIN {X 0,Y 334.219,Z 874.541,A -85,B 0,C 180,E1 -14925.073,E2 -14925.073} C_VEL
LIN {X 0,Y 332.972,Z 880.548,A -85,B 0,C 180,E1 -14926.575,E2 -14926.575} C_VEL
LIN {X 0,Y 331.593,Z 886.418,A -85,B 0,C 180,E1 -14928.384,E2 -14928.384} C_VEL
LIN {X 0,Y 330.855,Z 889.608,A -85,B 0,C 180,E1 -14929.598,E2 -14929.598} C_VEL
LIN {X 0,Y 329.695,Z 893.356,A -85,B 0,C 180,E1 -14931.418,E2 -14931.418} C_VEL
LIN {X 0,Y 329.053,Z 895.308,A -85,B 0,C 180,E1 -14932.637,E2 -14932.637} C_VEL
LIN {X 0,Y 328.193,Z 897.557,A -85,B 0,C 180,E1 -14935.086,E2 -14935.086} C_VEL
LIN {X 0,Y 327.876,Z 898.151,A -85,B 0,C 180,E1 -14936.313,E2 -14936.313} C_VEL
LIN {X 0,Y 327.517,Z 898.222,A -85,B 0,C 180,E1 -14937.54,E2 -14937.54} C_VEL
LIN {X 0,Y 327.298,Z 897.854,A -85,B 0,C 180,E1 -14938.77,E2 -14938.77} C_VEL
LIN {X 0,Y 326.959,Z 897.094,A -85,B 0,C 180,E1 -14940,E2 -14940} C_VEL
LIN {X 0,Y 326.93,Z 895.77,A -85,B 0,C 180,E1 -14941.232,E2 -14941.232} C_VEL
LIN {X 0,Y 326.608,Z 892.039,A -85,B 0,C 180,E1 -14943.701,E2 -14943.701} C_VEL
LIN {X 0,Y 326.997,Z 887.871,A -85,B 0,C 180,E1 -14945.55,E2 -14945.55} C_VEL
LIN {X 0,Y 327.302,Z 882.34,A -85,B 0,C 180,E1 -14947.448,E2 -14947.448} C_VEL
LIN {X 0,Y 327.635,Z 876.788,A -85,B 0,C 180,E1 -14949.005,E2 -14949.005} C_VEL
LIN {X 0,Y 327.973,Z 870.437,A -85,B 0,C 180,E1 -14950.495,E2 -14950.495} C_VEL
LIN {X 0,Y 328.477,Z 862.516,A -85,B 0,C 180,E1 -14952.041,E2 -14952.041} C_VEL
LIN {X 0,Y 328.983,Z 853.991,A -85,B 0,C 180,E1 -14953.434,E2 -14953.434} C_VEL
LIN {X 0,Y 329.496,Z 844.966,A -85,B 0,C 180,E1 -14954.672,E2 -14954.672} C_VEL
LIN {X 0,Y 330.024,Z 837.036,A -85,B 0,C 180,E1 -14955.596,E2 -14955.596} C_VEL
LIN {X 0,Y 330.472,Z 828.078,A -85,B 0,C 180,E1 -14956.486,E2 -14956.486} C_VEL
LIN {X 0,Y 330.933,Z 817.063,A -85,B 0,C 180,E1 -14957.376,E2 -14957.376} C_VEL
LIN {X 0,Y 331.271,Z 806.115,A -85,B 0,C 180,E1 -14958.076,E2 -14958.076} C_VEL
LIN {X 0,Y 331.486,Z 795.741,A -85,B 0,C 180,E1 -14958.584,E2 -14958.584} C_VEL
LIN {X 0,Y 331.671,Z 782.212,A -85,B 0,C 180,E1 -14959.054,E2 -14959.054} C_VEL
LIN {X 0,Y 332.88,Z 731.312,A -85,B 0,C 180,E1 -14960.524,E2 -14960.524} C_VEL
LIN {X 0,Y 326.672,Z 711.791,A -85,B 0,C 180,E1 -14961.383,E2 -14961.383} C_VEL
LIN {X 0,Y 326.657,Z 711.793,A -85,B 0,C 180,E1 -14965.487,E2 -14965.487} C_VEL
LIN {X 0,Y 326.611,Z 711.799,A -85,B 0,C 180,E1 -14969.664,E2 -14969.664} C_VEL
LIN {X 0,Y 326.637,Z 711.797,A -85,B 0,C 180,E1 -14972.942,E2 -14972.942} C_VEL
LIN {X 0,Y 326.632,Z 711.795,A -85,B 0,C 180,E1 -14975.517,E2 -14975.517} C_VEL
LIN {X 0,Y 326.593,Z 711.801,A -85,B 0,C 180,E1 -14979.215,E2 -14979.215} C_VEL
LIN {X 0,Y 326.592,Z 711.802,A -85,B 0,C 180,E1 -14982.967,E2 -14982.967} C_VEL
LIN {X 0,Y 326.592,Z 711.799,A -85,B 0,C 180,E1 -14987.026,E2 -14987.026} C_VEL
LIN {X 0,Y 326.591,Z 711.798,A -85,B 0,C 180,E1 -14990.778,E2 -14990.778} C_VEL
LIN {X 0,Y 326.629,Z 711.792,A -85,B 0,C 180,E1 -14994.475,E2 -14994.475} C_VEL
LIN {X 0,Y 326.621,Z 711.795,A -85,B 0,C 180,E1 -14997.45,E2 -14997.45} C_VEL
LIN {X 0,Y 326.593,Z 711.798,A -85,B 0,C 180,E1 -15000.327,E2 -15000.327} C_VEL
LIN {X 0,Y 326.611,Z 711.8,A -85,B 0,C 180,E1 -15003.129,E2 -15003.129} C_VEL
LIN {X 0,Y 326.666,Z 711.794,A -85,B 0,C 180,E1 -15005.759,E2 -15005.759} C_VEL
LIN {X 0,Y 327.831,Z 714.913,A -85,B 0,C 180,E1 -15005.939,E2 -15005.939} C_VEL
LIN {X 0,Y 337.841,Z 737.32,A -85,B 0,C 180,E1 -15007.242,E2 -15007.242} C_VEL
LIN {X 0,Y 337.128,Z 788.798,A -85,B 0,C 180,E1 -15008.358,E2 -15008.358} C_VEL
LIN {X 0,Y 337.039,Z 801.973,A -85,B 0,C 180,E1 -15008.775,E2 -15008.775} C_VEL
LIN {X 0,Y 336.631,Z 815.15,A -85,B 0,C 180,E1 -15009.445,E2 -15009.445} C_VEL
LIN {X 0,Y 335.876,Z 827.15,A -85,B 0,C 180,E1 -15010.29,E2 -15010.29} C_VEL
LIN {X 0,Y 334.928,Z 839.058,A -85,B 0,C 180,E1 -15011.415,E2 -15011.415} C_VEL
LIN {X 0,Y 333.766,Z 849.762,A -85,B 0,C 180,E1 -15012.69,E2 -15012.69} C_VEL
LIN {X 0,Y 332.704,Z 858.959,A -85,B 0,C 180,E1 -15014.054,E2 -15014.054} C_VEL
LIN {X 0,Y 331.619,Z 867.334,A -85,B 0,C 180,E1 -15015.573,E2 -15015.573} C_VEL
LIN {X 0,Y 330.365,Z 875.465,A -85,B 0,C 180,E1 -15017.398,E2 -15017.398} C_VEL
LIN {X 0,Y 329.338,Z 882.326,A -85,B 0,C 180,E1 -15019.337,E2 -15019.337} C_VEL
LIN {X 0,Y 328.603,Z 887.948,A -85,B 0,C 180,E1 -15021.382,E2 -15021.382} C_VEL
LIN {X 0,Y 327.828,Z 891.841,A -85,B 0,C 180,E1 -15023.221,E2 -15023.221} C_VEL
LIN {X 0,Y 327.292,Z 894.708,A -85,B 0,C 180,E1 -15025.065,E2 -15025.065} C_VEL
LIN {X 0,Y 327.173,Z 896.065,A -85,B 0,C 180,E1 -15026.297,E2 -15026.297} C_VEL
LIN {X 0,Y 327.138,Z 897.022,A -85,B 0,C 180,E1 -15027.529,E2 -15027.529} C_VEL
LIN {X 0,Y 326.938,Z 897.865,A -85,B 0,C 180,E1 -15029.992,E2 -15029.992} C_VEL
LIN {X 0,Y 327.14,Z 897.102,A -85,B 0,C 180,E1 -15032.454,E2 -15032.454} C_VEL
LIN {X 0,Y 327.275,Z 894.871,A -85,B 0,C 180,E1 -15034.919,E2 -15034.919} C_VEL
LIN {X 0,Y 327.815,Z 892.057,A -85,B 0,C 180,E1 -15036.763,E2 -15036.763} C_VEL
LIN {X 0,Y 328.579,Z 888.23,A -85,B 0,C 180,E1 -15038.602,E2 -15038.602} C_VEL
LIN {X 0,Y 329.308,Z 882.759,A -85,B 0,C 180,E1 -15040.636,E2 -15040.636} C_VEL
LIN {X 0,Y 330.344,Z 875.948,A -85,B 0,C 180,E1 -15042.586,E2 -15042.586} C_VEL
LIN {X 0,Y 331.59,Z 867.92,A -85,B 0,C 180,E1 -15044.411,E2 -15044.411} C_VEL
LIN {X 0,Y 332.661,Z 859.703,A -85,B 0,C 180,E1 -15045.931,E2 -15045.931} C_VEL
LIN {X 0,Y 333.817,Z 849.535,A -85,B 0,C 180,E1 -15047.449,E2 -15047.449} C_VEL
LIN {X 0,Y 335.008,Z 839.065,A -85,B 0,C 180,E1 -15048.69,E2 -15048.69} C_VEL
LIN {X 0,Y 335.99,Z 827.276,A -85,B 0,C 180,E1 -15049.801,E2 -15049.801} C_VEL
LIN {X 0,Y 336.739,Z 814.733,A -85,B 0,C 180,E1 -15050.683,E2 -15050.683} C_VEL
LIN {X 0,Y 337.106,Z 802.893,A -85,B 0,C 180,E1 -15051.29,E2 -15051.29} C_VEL
LIN {X 0,Y 337.225,Z 791.729,A -85,B 0,C 180,E1 -15051.671,E2 -15051.671} C_VEL
LIN {X 0,Y 337.614,Z 753.329,A -85,B 0,C 180,E1 -15052.521,E2 -15052.521} C_VEL
LIN {X 0,Y 337.87,Z 737.345,A -85,B 0,C 180,E1 -15052.866,E2 -15052.866} C_VEL
LIN {X 0,Y 334.729,Z 730.063,A -85,B 0,C 180,E1 -15053.272,E2 -15053.272} C_VEL
LIN {X 0,Y 332.463,Z 727.07,A -85,B 0,C 180,E1 -15053.517,E2 -15053.517} C_VEL
LIN {X 0,Y 322.957,Z 719.213,A -85,B 0,C 180,E1 -15054.477,E2 -15054.477} C_VEL
LIN {X 0,Y 320.974,Z 716.075,A -85,B 0,C 180,E1 -15054.722,E2 -15054.722} C_VEL
LIN {X 0,Y 319.691,Z 713.011,A -85,B 0,C 180,E1 -15054.908,E2 -15054.908} C_VEL
LIN {X 0,Y 319.634,Z 712.665,A -85,B 0,C 180,E1 -15054.943,E2 -15054.943} C_VEL
LIN {X 0,Y 319.554,Z 712.678,A -85,B 0,C 180,E1 -15058.925,E2 -15058.925} C_VEL
LIN {X 0,Y 319.501,Z 712.687,A -85,B 0,C 180,E1 -15061.853,E2 -15061.853} C_VEL
LIN {X 0,Y 319.547,Z 712.684,A -85,B 0,C 180,E1 -15065.534,E2 -15065.534} C_VEL
LIN {X 0,Y 319.546,Z 712.662,A -85,B 0,C 180,E1 -15067.998,E2 -15067.998} C_VEL
LIN {X 0,Y 319.562,Z 712.686,A -85,B 0,C 180,E1 -15071.604,E2 -15071.604} C_VEL
LIN {X 0,Y 319.602,Z 712.652,A -85,B 0,C 180,E1 -15075.277,E2 -15075.277} C_VEL
LIN {X 0,Y 319.536,Z 712.683,A -85,B 0,C 180,E1 -15078.713,E2 -15078.713} C_VEL
LIN {X 0,Y 319.531,Z 712.683,A -85,B 0,C 180,E1 -15082.336,E2 -15082.336} C_VEL
LIN {X 0,Y 319.507,Z 712.681,A -85,B 0,C 180,E1 -15085.116,E2 -15085.116} C_VEL
LIN {X 0,Y 319.518,Z 712.681,A -85,B 0,C 180,E1 -15089.051,E2 -15089.051} C_VEL
LIN {X 0,Y 319.55,Z 712.68,A -85,B 0,C 180,E1 -15092.492,E2 -15092.492} C_VEL
LIN {X 0,Y 319.543,Z 712.675,A -85,B 0,C 180,E1 -15095.299,E2 -15095.299} C_VEL
LIN {X 0,Y 319.534,Z 712.677,A -85,B 0,C 180,E1 -15098.043,E2 -15098.043} C_VEL
LIN {X 0,Y 319.626,Z 712.665,A -85,B 0,C 180,E1 -15100.958,E2 -15100.958} C_VEL
LIN {X 0,Y 319.665,Z 712.665,A -85,B 0,C 180,E1 -15105.273,E2 -15105.273} C_VEL
LIN {X 0,Y 319.69,Z 712.651,A -85,B 0,C 180,E1 -15109.871,E2 -15109.871} C_VEL
LIN {X 0,Y 319.853,Z 712.645,A -85,B 0,C 180,E1 -15112.424,E2 -15112.424} C_VEL
LIN {X 0,Y 319.685,Z 712.657,A -85,B 0,C 180,E1 -15114.955,E2 -15114.955} C_VEL
LIN {X 0,Y 319.948,Z 712.63,A -85,B 0,C 180,E1 -15117.482,E2 -15117.482} C_VEL
LIN {X 0,Y 320.099,Z 712.614,A -85,B 0,C 180,E1 -15120,E2 -15120} C_VEL
LIN {X 0,Y 319.949,Z 712.623,A -85,B 0,C 180,E1 -15122.518,E2 -15122.518} C_VEL
LIN {X 0,Y 319.879,Z 712.641,A -85,B 0,C 180,E1 -15126.307,E2 -15126.307} C_VEL
LIN {X 0,Y 319.772,Z 712.645,A -85,B 0,C 180,E1 -15128.85,E2 -15128.85} C_VEL
LIN {X 0,Y 319.616,Z 712.672,A -85,B 0,C 180,E1 -15132.703,E2 -15132.703} C_VEL
LIN {X 0,Y 319.634,Z 712.672,A -85,B 0,C 180,E1 -15135.299,E2 -15135.299} C_VEL
LIN {X 0,Y 319.588,Z 712.674,A -85,B 0,C 180,E1 -15139.26,E2 -15139.26} C_VEL
LIN {X 0,Y 319.5,Z 712.685,A -85,B 0,C 180,E1 -15143.325,E2 -15143.325} C_VEL
LIN {X 0,Y 319.559,Z 712.67,A -85,B 0,C 180,E1 -15146.095,E2 -15146.095} C_VEL
LIN {X 0,Y 319.532,Z 712.679,A -85,B 0,C 180,E1 -15148.939,E2 -15148.939} C_VEL
LIN {X 0,Y 319.482,Z 712.687,A -85,B 0,C 180,E1 -15151.867,E2 -15151.867} C_VEL
LIN {X 0,Y 319.527,Z 712.682,A -85,B 0,C 180,E1 -15155.55,E2 -15155.55} C_VEL
LIN {X 0,Y 319.533,Z 712.667,A -85,B 0,C 180,E1 -15158.014,E2 -15158.014} C_VEL
LIN {X 0,Y 319.554,Z 712.681,A -85,B 0,C 180,E1 -15161.62,E2 -15161.62} C_VEL
LIN {X 0,Y 319.602,Z 712.673,A -85,B 0,C 180,E1 -15165.293,E2 -15165.293} C_VEL
LIN {X 0,Y 319.543,Z 712.679,A -85,B 0,C 180,E1 -15168.729,E2 -15168.729} C_VEL
LIN {X 0,Y 319.581,Z 712.736,A -85,B 0,C 180,E1 -15171.556,E2 -15171.556} C_VEL
LIN {X 0,Y 322.795,Z 725.337,A -85,B 0,C 180,E1 -15174.731,E2 -15174.731} C_VEL
LIN {X 0,Y 325.601,Z 737.705,A -85,B 0,C 180,E1 -15177.658,E2 -15177.658} C_VEL
LIN {X 0,Y 326.966,Z 744.946,A -85,B 0,C 180,E1 -15179.293,E2 -15179.293} C_VEL
LIN {X 0,Y 324.253,Z 766.579,A -85,B 0,C 180,E1 -15183.631,E2 -15183.631} C_VEL
LIN {X 0,Y 323.515,Z 772.927,A -85,B 0,C 180,E1 -15184.896,E2 -15184.896} C_VEL
LIN {X 0,Y 327.439,Z 805.483,A -85,B 0,C 180,E1 -15185.965,E2 -15185.965} C_VEL
LIN {X 0,Y 329.868,Z 832.879,A -85,B 0,C 180,E1 -15186.777,E2 -15186.777} C_VEL
LIN {X 0,Y 328.592,Z 884.215,A -85,B 0,C 180,E1 -15187.906,E2 -15187.906} C_VEL
LIN {X 0,Y 327.792,Z 898.149,A -85,B 0,C 180,E1 -15188.469,E2 -15188.469} C_VEL
LIN {X 0,Y 326.572,Z 910.637,A -85,B 0,C 180,E1 -15189.211,E2 -15189.211} C_VEL
LIN {X 0,Y 325.25,Z 921.818,A -85,B 0,C 180,E1 -15190.113,E2 -15190.113} C_VEL
LIN {X 0,Y 323.704,Z 933.49,A -85,B 0,C 180,E1 -15191.333,E2 -15191.333} C_VEL
LIN {X 0,Y 322.207,Z 944.033,A -85,B 0,C 180,E1 -15192.721,E2 -15192.721} C_VEL
LIN {X 0,Y 321.143,Z 952.721,A -85,B 0,C 180,E1 -15194.135,E2 -15194.135} C_VEL
LIN {X 0,Y 320.328,Z 959.335,A -85,B 0,C 180,E1 -15195.417,E2 -15195.417} C_VEL
LIN {X 0,Y 319.354,Z 967.442,A -85,B 0,C 180,E1 -15197.296,E2 -15197.296} C_VEL
LIN {X 0,Y 318.778,Z 974.072,A -85,B 0,C 180,E1 -15199.208,E2 -15199.208} C_VEL
LIN {X 0,Y 318.577,Z 979.382,A -85,B 0,C 180,E1 -15201.126,E2 -15201.126} C_VEL
LIN {X 0,Y 318.623,Z 983.503,A -85,B 0,C 180,E1 -15203.019,E2 -15203.019} C_VEL
LIN {X 0,Y 318.809,Z 986.641,A -85,B 0,C 180,E1 -15204.95,E2 -15204.95} C_VEL
LIN {X 0,Y 318.964,Z 988.123,A -85,B 0,C 180,E1 -15206.219,E2 -15206.219} C_VEL
LIN {X 0,Y 319.014,Z 989.17,A -85,B 0,C 180,E1 -15207.483,E2 -15207.483} C_VEL
LIN {X 0,Y 319.114,Z 989.817,A -85,B 0,C 180,E1 -15208.747,E2 -15208.747} C_VEL
LIN {X 0,Y 319.206,Z 990.05,A -85,B 0,C 180,E1 -15210.008,E2 -15210.008} C_VEL
LIN {X 0,Y 319.114,Z 989.805,A -85,B 0,C 180,E1 -15211.27,E2 -15211.27} C_VEL
LIN {X 0,Y 319.016,Z 989.149,A -85,B 0,C 180,E1 -15212.534,E2 -15212.534} C_VEL
LIN {X 0,Y 318.964,Z 988.092,A -85,B 0,C 180,E1 -15213.798,E2 -15213.798} C_VEL
LIN {X 0,Y 318.786,Z 986.593,A -85,B 0,C 180,E1 -15215.067,E2 -15215.067} C_VEL
LIN {X 0,Y 318.616,Z 983.496,A -85,B 0,C 180,E1 -15216.971,E2 -15216.971} C_VEL
LIN {X 0,Y 318.589,Z 979.313,A -85,B 0,C 180,E1 -15218.891,E2 -15218.891} C_VEL
LIN {X 0,Y 318.844,Z 972.938,A -85,B 0,C 180,E1 -15221.128,E2 -15221.128} C_VEL
LIN {X 0,Y 319.488,Z 966.062,A -85,B 0,C 180,E1 -15223.039,E2 -15223.039} C_VEL
LIN {X 0,Y 320.604,Z 956.346,A -85,B 0,C 180,E1 -15225.259,E2 -15225.259} C_VEL
LIN {X 0,Y 321.869,Z 948.178,A -85,B 0,C 180,E1 -15226.824,E2 -15226.824} C_VEL
LIN {X 0,Y 323.303,Z 939.49,A -85,B 0,C 180,E1 -15228.216,E2 -15228.216} C_VEL
LIN {X 0,Y 324.986,Z 929.158,A -85,B 0,C 180,E1 -15229.592,E2 -15229.592} C_VEL
LIN {X 0,Y 326.619,Z 919.678,A -85,B 0,C 180,E1 -15230.638,E2 -15230.638} C_VEL
LIN {X 0,Y 328.178,Z 910.036,A -85,B 0,C 180,E1 -15231.522,E2 -15231.522} C_VEL
LIN {X 0,Y 329.734,Z 899.319,A -85,B 0,C 180,E1 -15232.32,E2 -15232.32} C_VEL
LIN {X 0,Y 331.179,Z 887.709,A -85,B 0,C 180,E1 -15232.999,E2 -15232.999} C_VEL
LIN {X 0,Y 332.222,Z 876.738,A -85,B 0,C 180,E1 -15233.5,E2 -15233.5} C_VEL
LIN {X 0,Y 335.227,Z 832.122,A -85,B 0,C 180,E1 -15235.041,E2 -15235.041} C_VEL
LIN {X 0,Y 334.515,Z 805.797,A -85,B 0,C 180,E1 -15236.352,E2 -15236.352} C_VEL
LIN {X 0,Y 333.03,Z 788.005,A -85,B 0,C 180,E1 -15237.461,E2 -15237.461} C_VEL
LIN {X 0,Y 331.013,Z 770.16,A -85,B 0,C 180,E1 -15238.745,E2 -15238.745} C_VEL
LIN {X 0,Y 329.285,Z 757.538,A -85,B 0,C 180,E1 -15239.779,E2 -15239.779} C_VEL
LIN {X 0,Y 328.066,Z 749.373,A -85,B 0,C 180,E1 -15240.515,E2 -15240.515} C_VEL
LIN {X 0,Y 327.192,Z 744.45,A -85,B 0,C 180,E1 -15241.158,E2 -15241.158} C_VEL
LIN {X 0,Y 325.812,Z 738.638,A -85,B 0,C 180,E1 -15242.106,E2 -15242.106} C_VEL
LIN {X 0,Y 322.791,Z 725.258,A -85,B 0,C 180,E1 -15245.267,E2 -15245.267} C_VEL
LIN {X 0,Y 319.553,Z 712.678,A -85,B 0,C 180,E1 -15248.47,E2 -15248.47} C_VEL
LIN {X 0,Y 319.512,Z 712.686,A -85,B 0,C 180,E1 -15251.594,E2 -15251.594} C_VEL
LIN {X 0,Y 319.5,Z 712.684,A -85,B 0,C 180,E1 -15254.749,E2 -15254.749} C_VEL
LIN {X 0,Y 319.514,Z 712.682,A -85,B 0,C 180,E1 -15258.413,E2 -15258.413} C_VEL
LIN {X 0,Y 319.561,Z 712.676,A -85,B 0,C 180,E1 -15262.356,E2 -15262.356} C_VEL
LIN {X 0,Y 319.58,Z 712.675,A -85,B 0,C 180,E1 -15265.126,E2 -15265.126} C_VEL
LIN {X 0,Y 319.617,Z 712.867,A -85,B 0,C 180,E1 -15267.314,E2 -15267.314} C_VEL
LIN {X 0,Y 320.479,Z 715.37,A -85,B 0,C 180,E1 -15267.824,E2 -15267.824} C_VEL
LIN {X 0,Y 322.54,Z 717.639,A -85,B 0,C 180,E1 -15268.641,E2 -15268.641} C_VEL
LIN {X 0,Y 323.484,Z 718.454,A -85,B 0,C 180,E1 -15268.981,E2 -15268.981} C_VEL
LIN {X 0,Y 325.043,Z 721.365,A -85,B 0,C 180,E1 -15269.629,E2 -15269.629} C_VEL
LIN {X 0,Y 326.846,Z 723.439,A -85,B 0,C 180,E1 -15270.242,E2 -15270.242} C_VEL
LIN {X 0,Y 328.956,Z 726.766,A -85,B 0,C 180,E1 -15270.977,E2 -15270.977} C_VEL
LIN {X 0,Y 330.371,Z 728.87,A -85,B 0,C 180,E1 -15271.427,E2 -15271.427} C_VEL
LIN {X 0,Y 334.542,Z 735.574,A -85,B 0,C 180,E1 -15272.701,E2 -15272.701} C_VEL
LIN {X 0,Y 339.106,Z 744.061,A -85,B 0,C 180,E1 -15274.005,E2 -15274.005} C_VEL
LIN {X 0,Y 340.48,Z 747.058,A -85,B 0,C 180,E1 -15274.385,E2 -15274.385} C_VEL
LIN {X 0,Y 337.052,Z 791.16,A -85,B 0,C 180,E1 -15275.968,E2 -15275.968} C_VEL
LIN {X 0,Y 336.442,Z 807.557,A -85,B 0,C 180,E1 -15276.66,E2 -15276.66} C_VEL
LIN {X 0,Y 335.786,Z 818.853,A -85,B 0,C 180,E1 -15277.298,E2 -15277.298} C_VEL
LIN {X 0,Y 334.838,Z 829.985,A -85,B 0,C 180,E1 -15278.115,E2 -15278.115} C_VEL
LIN {X 0,Y 333.624,Z 841.476,A -85,B 0,C 180,E1 -15279.177,E2 -15279.177} C_VEL
LIN {X 0,Y 332.005,Z 852.944,A -85,B 0,C 180,E1 -15280.525,E2 -15280.525} C_VEL
LIN {X 0,Y 330.777,Z 861.169,A -85,B 0,C 180,E1 -15281.736,E2 -15281.736} C_VEL
LIN {X 0,Y 329.488,Z 868.183,A -85,B 0,C 180,E1 -15282.945,E2 -15282.945} C_VEL
LIN {X 0,Y 327.985,Z 875.533,A -85,B 0,C 180,E1 -15284.464,E2 -15284.464} C_VEL
LIN {X 0,Y 326.743,Z 881.208,A -85,B 0,C 180,E1 -15285.876,E2 -15285.876} C_VEL
LIN {X 0,Y 325.388,Z 886.623,A -85,B 0,C 180,E1 -15287.526,E2 -15287.526} C_VEL
LIN {X 0,Y 324.431,Z 890.025,A -85,B 0,C 180,E1 -15288.757,E2 -15288.757} C_VEL
LIN {X 0,Y 323.319,Z 893.963,A -85,B 0,C 180,E1 -15290.617,E2 -15290.617} C_VEL
LIN {X 0,Y 322.194,Z 896.833,A -85,B 0,C 180,E1 -15292.48,E2 -15292.48} C_VEL
LIN {X 0,Y 321.698,Z 898.09,A -85,B 0,C 180,E1 -15293.729,E2 -15293.729} C_VEL
LIN {X 0,Y 320.917,Z 899.399,A -85,B 0,C 180,E1 -15296.233,E2 -15296.233} C_VEL
LIN {X 0,Y 320.529,Z 899.384,A -85,B 0,C 180,E1 -15297.487,E2 -15297.487} C_VEL
LIN {X 0,Y 320.3,Z 898.944,A -85,B 0,C 180,E1 -15298.743,E2 -15298.743} C_VEL
LIN {X 0,Y 319.932,Z 898.063,A -85,B 0,C 180,E1 -15300,E2 -15300} C_VEL
LIN {X 0,Y 319.905,Z 896.687,A -85,B 0,C 180,E1 -15301.259,E2 -15301.259} C_VEL
LIN {X 0,Y 319.558,Z 892.698,A -85,B 0,C 180,E1 -15303.783,E2 -15303.783} C_VEL
LIN {X 0,Y 319.966,Z 888.358,A -85,B 0,C 180,E1 -15305.673,E2 -15305.673} C_VEL
LIN {X 0,Y 320.241,Z 883.149,A -85,B 0,C 180,E1 -15307.468,E2 -15307.468} C_VEL
LIN {X 0,Y 320.602,Z 877.369,A -85,B 0,C 180,E1 -15309.097,E2 -15309.097} C_VEL
LIN {X 0,Y 320.957,Z 870.412,A -85,B 0,C 180,E1 -15310.727,E2 -15310.727} C_VEL
LIN {X 0,Y 321.398,Z 864.078,A -85,B 0,C 180,E1 -15311.99,E2 -15311.99} C_VEL
LIN {X 0,Y 321.883,Z 855.635,A -85,B 0,C 180,E1 -15313.414,E2 -15313.414} C_VEL
LIN {X 0,Y 322.446,Z 846.704,A -85,B 0,C 180,E1 -15314.678,E2 -15314.678} C_VEL
LIN {X 0,Y 323.028,Z 837.409,A -85,B 0,C 180,E1 -15315.781,E2 -15315.781} C_VEL
LIN {X 0,Y 323.538,Z 827.378,A -85,B 0,C 180,E1 -15316.771,E2 -15316.771} C_VEL
LIN {X 0,Y 323.939,Z 817.335,A -85,B 0,C 180,E1 -15317.583,E2 -15317.583} C_VEL
LIN {X 0,Y 324.273,Z 807.304,A -85,B 0,C 180,E1 -15318.235,E2 -15318.235} C_VEL
LIN {X 0,Y 324.504,Z 797.023,A -85,B 0,C 180,E1 -15318.753,E2 -15318.753} C_VEL
LIN {X 0,Y 324.703,Z 783.686,A -85,B 0,C 180,E1 -15319.233,E2 -15319.233} C_VEL
LIN {X 0,Y 325.81,Z 732.216,A -85,B 0,C 180,E1 -15320.766,E2 -15320.766} C_VEL
LIN {X 0,Y 319.634,Z 712.667,A -85,B 0,C 180,E1 -15321.683,E2 -15321.683} C_VEL
LIN {X 0,Y 319.593,Z 712.673,A -85,B 0,C 180,E1 -15326.092,E2 -15326.092} C_VEL
LIN {X 0,Y 319.554,Z 712.682,A -85,B 0,C 180,E1 -15328.937,E2 -15328.937} C_VEL
LIN {X 0,Y 319.544,Z 712.679,A -85,B 0,C 180,E1 -15331.861,E2 -15331.861} C_VEL
LIN {X 0,Y 319.6,Z 712.671,A -85,B 0,C 180,E1 -15335.539,E2 -15335.539} C_VEL
LIN {X 0,Y 319.551,Z 712.676,A -85,B 0,C 180,E1 -15339.659,E2 -15339.659} C_VEL
LIN {X 0,Y 319.539,Z 712.676,A -85,B 0,C 180,E1 -15343.456,E2 -15343.456} C_VEL
LIN {X 0,Y 319.571,Z 712.673,A -85,B 0,C 180,E1 -15347.012,E2 -15347.012} C_VEL
LIN {X 0,Y 319.536,Z 712.676,A -85,B 0,C 180,E1 -15350.362,E2 -15350.362} C_VEL
LIN {X 0,Y 319.597,Z 712.668,A -85,B 0,C 180,E1 -15354.453,E2 -15354.453} C_VEL
LIN {X 0,Y 319.537,Z 712.676,A -85,B 0,C 180,E1 -15358.131,E2 -15358.131} C_VEL
LIN {X 0,Y 319.56,Z 712.676,A -85,B 0,C 180,E1 -15361.608,E2 -15361.608} C_VEL
LIN {X 0,Y 319.615,Z 712.725,A -85,B 0,C 180,E1 -15365.194,E2 -15365.194} C_VEL
LIN {X 0,Y 320.729,Z 715.695,A -85,B 0,C 180,E1 -15365.363,E2 -15365.363} C_VEL
LIN {X 0,Y 329.33,Z 734.417,A -85,B 0,C 180,E1 -15366.52,E2 -15366.52} C_VEL
LIN {X 0,Y 331.31,Z 739.065,A -85,B 0,C 180,E1 -15366.784,E2 -15366.784} C_VEL
LIN {X 0,Y 330.582,Z 789.026,A -85,B 0,C 180,E1 -15367.888,E2 -15367.888} C_VEL
LIN {X 0,Y 330.497,Z 802.402,A -85,B 0,C 180,E1 -15368.307,E2 -15368.307} C_VEL
LIN {X 0,Y 330.132,Z 814.873,A -85,B 0,C 180,E1 -15368.939,E2 -15368.939} C_VEL
LIN {X 0,Y 329.406,Z 826.406,A -85,B 0,C 180,E1 -15369.74,E2 -15369.74} C_VEL
LIN {X 0,Y 328.462,Z 837.99,A -85,B 0,C 180,E1 -15370.797,E2 -15370.797} C_VEL
LIN {X 0,Y 327.335,Z 848.462,A -85,B 0,C 180,E1 -15372.016,E2 -15372.016} C_VEL
LIN {X 0,Y 326.146,Z 858.061,A -85,B 0,C 180,E1 -15373.403,E2 -15373.403} C_VEL
LIN {X 0,Y 325.079,Z 866.757,A -85,B 0,C 180,E1 -15374.956,E2 -15374.956} C_VEL
LIN {X 0,Y 323.721,Z 875.261,A -85,B 0,C 180,E1 -15376.816,E2 -15376.816} C_VEL
LIN {X 0,Y 322.581,Z 882.025,A -85,B 0,C 180,E1 -15378.684,E2 -15378.684} C_VEL
LIN {X 0,Y 321.93,Z 887.391,A -85,B 0,C 180,E1 -15380.569,E2 -15380.569} C_VEL
LIN {X 0,Y 321.492,Z 890.328,A -85,B 0,C 180,E1 -15381.823,E2 -15381.823} C_VEL
LIN {X 0,Y 320.622,Z 893.888,A -85,B 0,C 180,E1 -15383.7,E2 -15383.7} C_VEL
LIN {X 0,Y 320.29,Z 895.712,A -85,B 0,C 180,E1 -15384.957,E2 -15384.957} C_VEL
LIN {X 0,Y 320.118,Z 898.025,A -85,B 0,C 180,E1 -15387.475,E2 -15387.475} C_VEL
LIN {X 0,Y 319.911,Z 898.867,A -85,B 0,C 180,E1 -15389.992,E2 -15389.992} C_VEL
LIN {X 0,Y 320.119,Z 898.104,A -85,B 0,C 180,E1 -15392.508,E2 -15392.508} C_VEL
LIN {X 0,Y 320.273,Z 895.874,A -85,B 0,C 180,E1 -15395.027,E2 -15395.027} C_VEL
LIN {X 0,Y 320.839,Z 893.058,A -85,B 0,C 180,E1 -15396.911,E2 -15396.911} C_VEL
LIN {X 0,Y 321.634,Z 889.231,A -85,B 0,C 180,E1 -15398.789,E2 -15398.789} C_VEL
LIN {X 0,Y 322.404,Z 883.76,A -85,B 0,C 180,E1 -15400.866,E2 -15400.866} C_VEL
LIN {X 0,Y 323.488,Z 876.948,A -85,B 0,C 180,E1 -15402.858,E2 -15402.858} C_VEL
LIN {X 0,Y 324.788,Z 868.92,A -85,B 0,C 180,E1 -15404.72,E2 -15404.72} C_VEL
LIN {X 0,Y 325.908,Z 860.702,A -85,B 0,C 180,E1 -15406.271,E2 -15406.271} C_VEL
LIN {X 0,Y 327.119,Z 850.534,A -85,B 0,C 180,E1 -15407.818,E2 -15407.818} C_VEL
LIN {X 0,Y 328.348,Z 840.064,A -85,B 0,C 180,E1 -15409.083,E2 -15409.083} C_VEL
LIN {X 0,Y 329.337,Z 828.8,A -85,B 0,C 180,E1 -15410.17,E2 -15410.17} C_VEL
LIN {X 0,Y 330.153,Z 816.881,A -85,B 0,C 180,E1 -15411.042,E2 -15411.042} C_VEL
LIN {X 0,Y 330.511,Z 804.943,A -85,B 0,C 180,E1 -15411.689,E2 -15411.689} C_VEL
LIN {X 0,Y 330.663,Z 793.259,A -85,B 0,C 180,E1 -15412.108,E2 -15412.108} C_VEL
LIN {X 0,Y 331.032,Z 759.377,A -85,B 0,C 180,E1 -15412.877,E2 -15412.877} C_VEL
LIN {X 0,Y 331.368,Z 739.11,A -85,B 0,C 180,E1 -15413.323,E2 -15413.323} C_VEL
LIN {X 0,Y 321.918,Z 718.181,A -85,B 0,C 180,E1 -15414.59,E2 -15414.59} C_VEL
LIN {X 0,Y 320.974,Z 716.075,A -85,B 0,C 180,E1 -15414.722,E2 -15414.722} C_VEL
LIN {X 0,Y 319.893,Z 714.284,A -85,B 0,C 180,E1 -15414.963,E2 -15414.963} C_VEL
LIN {X 0,Y 318.309,Z 713.086,A -85,B 0,C 180,E1 -15415.469,E2 -15415.469} C_VEL
LIN {X 0,Y 316.445,Z 713.059,A -85,B 0,C 180,E1 -15416.257,E2 -15416.257} C_VEL
LIN {X 0,Y 314.114,Z 713.488,A -85,B 0,C 180,E1 -15417.721,E2 -15417.721} C_VEL
LIN {X 0,Y 312.694,Z 713.574,A -85,B 0,C 180,E1 -15419.355,E2 -15419.355} C_VEL
LIN {X 0,Y 312.48,Z 713.556,A -85,B 0,C 180,E1 -15420.183,E2 -15420.183} C_VEL
LIN {X 0,Y 312.474,Z 713.558,A -85,B 0,C 180,E1 -15424.201,E2 -15424.201} C_VEL
LIN {X 0,Y 312.507,Z 713.539,A -85,B 0,C 180,E1 -15428.083,E2 -15428.083} C_VEL
LIN {X 0,Y 312.516,Z 713.559,A -85,B 0,C 180,E1 -15432.087,E2 -15432.087} C_VEL
LIN {X 0,Y 312.551,Z 713.532,A -85,B 0,C 180,E1 -15435.808,E2 -15435.808} C_VEL
LIN {X 0,Y 312.483,Z 713.561,A -85,B 0,C 180,E1 -15439.861,E2 -15439.861} C_VEL
LIN {X 0,Y 312.489,Z 713.559,A -85,B 0,C 180,E1 -15442.61,E2 -15442.61} C_VEL
LIN {X 0,Y 312.466,Z 713.556,A -85,B 0,C 180,E1 -15446.304,E2 -15446.304} C_VEL
LIN {X 0,Y 312.489,Z 713.55,A -85,B 0,C 180,E1 -15450.344,E2 -15450.344} C_VEL
LIN {X 0,Y 312.543,Z 713.555,A -85,B 0,C 180,E1 -15454.06,E2 -15454.06} C_VEL
LIN {X 0,Y 312.525,Z 713.547,A -85,B 0,C 180,E1 -15457.524,E2 -15457.524} C_VEL
LIN {X 0,Y 312.574,Z 713.542,A -85,B 0,C 180,E1 -15461.652,E2 -15461.652} C_VEL
LIN {X 0,Y 312.627,Z 713.542,A -85,B 0,C 180,E1 -15465.683,E2 -15465.683} C_VEL
LIN {X 0,Y 312.635,Z 713.529,A -85,B 0,C 180,E1 -15469.64,E2 -15469.64} C_VEL
LIN {X 0,Y 312.793,Z 713.523,A -85,B 0,C 180,E1 -15472.252,E2 -15472.252} C_VEL
LIN {X 0,Y 312.655,Z 713.534,A -85,B 0,C 180,E1 -15474.841,E2 -15474.841} C_VEL
LIN {X 0,Y 312.892,Z 713.508,A -85,B 0,C 180,E1 -15477.425,E2 -15477.425} C_VEL
LIN {X 0,Y 313.051,Z 713.492,A -85,B 0,C 180,E1 -15480,E2 -15480} C_VEL
LIN {X 0,Y 312.892,Z 713.501,A -85,B 0,C 180,E1 -15482.575,E2 -15482.575} C_VEL
LIN {X 0,Y 312.837,Z 713.519,A -85,B 0,C 180,E1 -15486.449,E2 -15486.449} C_VEL
LIN {X 0,Y 312.719,Z 713.522,A -85,B 0,C 180,E1 -15489.051,E2 -15489.051} C_VEL
LIN {X 0,Y 312.568,Z 713.552,A -85,B 0,C 180,E1 -15492.994,E2 -15492.994} C_VEL
LIN {X 0,Y 312.573,Z 713.55,A -85,B 0,C 180,E1 -15495.653,E2 -15495.653} C_VEL
LIN {X 0,Y 312.545,Z 713.552,A -85,B 0,C 180,E1 -15499.229,E2 -15499.229} C_VEL
LIN {X 0,Y 312.466,Z 713.559,A -85,B 0,C 180,E1 -15502.786,E2 -15502.786} C_VEL
LIN {X 0,Y 312.537,Z 713.544,A -85,B 0,C 180,E1 -15505.938,E2 -15505.938} C_VEL
LIN {X 0,Y 312.489,Z 713.555,A -85,B 0,C 180,E1 -15509.656,E2 -15509.656} C_VEL
LIN {X 0,Y 312.466,Z 713.559,A -85,B 0,C 180,E1 -15513.695,E2 -15513.695} C_VEL
LIN {X 0,Y 312.49,Z 713.552,A -85,B 0,C 180,E1 -15517.39,E2 -15517.39} C_VEL
LIN {X 0,Y 312.48,Z 713.559,A -85,B 0,C 180,E1 -15520.711,E2 -15520.711} C_VEL
LIN {X 0,Y 312.55,Z 713.554,A -85,B 0,C 180,E1 -15524.192,E2 -15524.192} C_VEL
LIN {X 0,Y 312.515,Z 713.547,A -85,B 0,C 180,E1 -15527.913,E2 -15527.913} C_VEL
LIN {X 0,Y 312.544,Z 713.616,A -85,B 0,C 180,E1 -15530.992,E2 -15530.992} C_VEL
LIN {X 0,Y 315.897,Z 726.657,A -85,B 0,C 180,E1 -15534.381,E2 -15534.381} C_VEL
LIN {X 0,Y 318.365,Z 737.473,A -85,B 0,C 180,E1 -15537.02,E2 -15537.02} C_VEL
LIN {X 0,Y 320.106,Z 746.639,A -85,B 0,C 180,E1 -15539.15,E2 -15539.15} C_VEL
LIN {X 0,Y 317.36,Z 767.172,A -85,B 0,C 180,E1 -15543.368,E2 -15543.368} C_VEL
LIN {X 0,Y 316.823,Z 772.091,A -85,B 0,C 180,E1 -15544.332,E2 -15544.332} C_VEL
LIN {X 0,Y 320.873,Z 805.621,A -85,B 0,C 180,E1 -15545.468,E2 -15545.468} C_VEL
LIN {X 0,Y 323.32,Z 832.826,A -85,B 0,C 180,E1 -15546.3,E2 -15546.3} C_VEL
LIN {X 0,Y 322.016,Z 883.215,A -85,B 0,C 180,E1 -15547.43,E2 -15547.43} C_VEL
LIN {X 0,Y 321.168,Z 897.14,A -85,B 0,C 180,E1 -15548.002,E2 -15548.002} C_VEL
LIN {X 0,Y 319.899,Z 909.623,A -85,B 0,C 180,E1 -15548.757,E2 -15548.757} C_VEL
LIN {X 0,Y 318.562,Z 920.806,A -85,B 0,C 180,E1 -15549.678,E2 -15549.678} C_VEL
LIN {X 0,Y 316.961,Z 932.477,A -85,B 0,C 180,E1 -15550.92,E2 -15550.92} C_VEL
LIN {X 0,Y 315.362,Z 943.013,A -85,B 0,C 180,E1 -15552.334,E2 -15552.334} C_VEL
LIN {X 0,Y 314.264,Z 951.698,A -85,B 0,C 180,E1 -15553.777,E2 -15553.777} C_VEL
LIN {X 0,Y 313.289,Z 958.727,A -85,B 0,C 180,E1 -15555.174,E2 -15555.174} C_VEL
LIN {X 0,Y 312.37,Z 966.422,A -85,B 0,C 180,E1 -15557.007,E2 -15557.007} C_VEL
LIN {X 0,Y 311.729,Z 973.049,A -85,B 0,C 180,E1 -15558.961,E2 -15558.961} C_VEL
LIN {X 0,Y 311.516,Z 978.363,A -85,B 0,C 180,E1 -15560.923,E2 -15560.923} C_VEL
LIN {X 0,Y 311.553,Z 982.739,A -85,B 0,C 180,E1 -15563.004,E2 -15563.004} C_VEL
LIN {X 0,Y 311.74,Z 985.629,A -85,B 0,C 180,E1 -15564.835,E2 -15564.835} C_VEL
LIN {X 0,Y 311.919,Z 987.116,A -85,B 0,C 180,E1 -15566.133,E2 -15566.133} C_VEL
LIN {X 0,Y 311.97,Z 988.164,A -85,B 0,C 180,E1 -15567.426,E2 -15567.426} C_VEL
LIN {X 0,Y 312.075,Z 988.813,A -85,B 0,C 180,E1 -15568.718,E2 -15568.718} C_VEL
LIN {X 0,Y 312.175,Z 989.047,A -85,B 0,C 180,E1 -15570.009,E2 -15570.009} C_VEL
LIN {X 0,Y 312.075,Z 988.8,A -85,B 0,C 180,E1 -15571.299,E2 -15571.299} C_VEL
LIN {X 0,Y 311.971,Z 988.142,A -85,B 0,C 180,E1 -15572.591,E2 -15572.591} C_VEL
LIN {X 0,Y 311.917,Z 987.084,A -85,B 0,C 180,E1 -15573.884,E2 -15573.884} C_VEL
LIN {X 0,Y 311.719,Z 985.58,A -85,B 0,C 180,E1 -15575.182,E2 -15575.182} C_VEL
LIN {X 0,Y 311.547,Z 982.727,A -85,B 0,C 180,E1 -15576.987,E2 -15576.987} C_VEL
LIN {X 0,Y 311.527,Z 978.292,A -85,B 0,C 180,E1 -15579.094,E2 -15579.094} C_VEL
LIN {X 0,Y 311.84,Z 971.917,A -85,B 0,C 180,E1 -15581.381,E2 -15581.381} C_VEL
LIN {X 0,Y 312.849,Z 962.993,A -85,B 0,C 180,E1 -15583.983,E2 -15583.983} C_VEL
LIN {X 0,Y 313.763,Z 956.229,A -85,B 0,C 180,E1 -15585.6,E2 -15585.6} C_VEL
LIN {X 0,Y 315.306,Z 946.433,A -85,B 0,C 180,E1 -15587.52,E2 -15587.52} C_VEL
LIN {X 0,Y 316.949,Z 937.751,A -85,B 0,C 180,E1 -15588.93,E2 -15588.93} C_VEL
LIN {X 0,Y 318.593,Z 928.681,A -85,B 0,C 180,E1 -15590.17,E2 -15590.17} C_VEL
LIN {X 0,Y 320.317,Z 919.332,A -85,B 0,C 180,E1 -15591.232,E2 -15591.232} C_VEL
LIN {X 0,Y 322.206,Z 908.238,A -85,B 0,C 180,E1 -15592.278,E2 -15592.278} C_VEL
LIN {X 0,Y 323.917,Z 897.59,A -85,B 0,C 180,E1 -15593.08,E2 -15593.08} C_VEL
LIN {X 0,Y 325.426,Z 886.117,A -85,B 0,C 180,E1 -15593.767,E2 -15593.767} C_VEL
LIN {X 0,Y 326.564,Z 875.23,A -85,B 0,C 180,E1 -15594.265,E2 -15594.265} C_VEL
LIN {X 0,Y 329.675,Z 832.822,A -85,B 0,C 180,E1 -15595.792,E2 -15595.792} C_VEL
LIN {X 0,Y 329.196,Z 807.886,A -85,B 0,C 180,E1 -15597.082,E2 -15597.082} C_VEL
LIN {X 0,Y 327.755,Z 788.368,A -85,B 0,C 180,E1 -15598.347,E2 -15598.347} C_VEL
LIN {X 0,Y 325.895,Z 770.585,A -85,B 0,C 180,E1 -15599.703,E2 -15599.703} C_VEL
LIN {X 0,Y 324.612,Z 760.058,A -85,B 0,C 180,E1 -15600.616,E2 -15600.616} C_VEL
LIN {X 0,Y 323.518,Z 751.861,A -85,B 0,C 180,E1 -15601.38,E2 -15601.38} C_VEL
LIN {X 0,Y 321.985,Z 746.156,A -85,B 0,C 180,E1 -15602.146,E2 -15602.146} C_VEL
LIN {X 0,Y 320.577,Z 740.84,A -85,B 0,C 180,E1 -15603.133,E2 -15603.133} C_VEL
LIN {X 0,Y 317.608,Z 729.899,A -85,B 0,C 180,E1 -15605.552,E2 -15605.552} C_VEL
LIN {X 0,Y 315.663,Z 720.275,A -85,B 0,C 180,E1 -15608.152,E2 -15608.152} C_VEL
LIN {X 0,Y 315.354,Z 718.413,A -85,B 0,C 180,E1 -15608.738,E2 -15608.738} C_VEL
LIN {X 0,Y 313.231,Z 715.991,A -85,B 0,C 180,E1 -15610.6,E2 -15610.6} C_VEL
LIN {X 0,Y 312.442,Z 713.563,A -85,B 0,C 180,E1 -15612.208,E2 -15612.208} C_VEL
LIN {X 0,Y 312.473,Z 713.56,A -85,B 0,C 180,E1 -15616.04,E2 -15616.04} C_VEL
LIN {X 0,Y 312.458,Z 713.564,A -85,B 0,C 180,E1 -15619.893,E2 -15619.893} C_VEL
LIN {X 0,Y 312.552,Z 713.551,A -85,B 0,C 180,E1 -15624.055,E2 -15624.055} C_VEL
LIN {X 0,Y 312.744,Z 714.503,A -85,B 0,C 180,E1 -15624.722,E2 -15624.722} C_VEL
LIN {X 0,Y 314.023,Z 717.073,A -85,B 0,C 180,E1 -15625.594,E2 -15625.594} C_VEL
LIN {X 0,Y 316.323,Z 718.958,A -85,B 0,C 180,E1 -15626.706,E2 -15626.706} C_VEL
LIN {X 0,Y 316.838,Z 719.738,A -85,B 0,C 180,E1 -15626.964,E2 -15626.964} C_VEL
LIN {X 0,Y 318.552,Z 722.764,A -85,B 0,C 180,E1 -15627.824,E2 -15627.824} C_VEL
LIN {X 0,Y 320.532,Z 724.867,A -85,B 0,C 180,E1 -15628.615,E2 -15628.615} C_VEL
LIN {X 0,Y 322.679,Z 728.2,A -85,B 0,C 180,E1 -15629.502,E2 -15629.502} C_VEL
LIN {X 0,Y 324.031,Z 730.223,A -85,B 0,C 180,E1 -15629.999,E2 -15629.999} C_VEL
LIN {X 0,Y 326.973,Z 734.752,A -85,B 0,C 180,E1 -15631.038,E2 -15631.038} C_VEL
LIN {X 0,Y 330.956,Z 741.459,A -85,B 0,C 180,E1 -15632.335,E2 -15632.335} C_VEL
LIN {X 0,Y 335.029,Z 749.316,A -85,B 0,C 180,E1 -15633.559,E2 -15633.559} C_VEL
LIN {X 0,Y 335.214,Z 749.931,A -85,B 0,C 180,E1 -15633.627,E2 -15633.627} C_VEL
LIN {X 0,Y 331.633,Z 793.502,A -85,B 0,C 180,E1 -15635.245,E2 -15635.245} C_VEL
LIN {X 0,Y 330.866,Z 810.129,A -85,B 0,C 180,E1 -15635.996,E2 -15635.996} C_VEL
LIN {X 0,Y 330.005,Z 822.408,A -85,B 0,C 180,E1 -15636.728,E2 -15636.728} C_VEL
LIN {X 0,Y 328.885,Z 834.828,A -85,B 0,C 180,E1 -15637.71,E2 -15637.71} C_VEL
LIN {X 0,Y 327.357,Z 846.555,A -85,B 0,C 180,E1 -15638.924,E2 -15638.924} C_VEL
LIN {X 0,Y 325.978,Z 855.012,A -85,B 0,C 180,E1 -15639.985,E2 -15639.985} C_VEL
LIN {X 0,Y 324.826,Z 862.211,A -85,B 0,C 180,E1 -15641.062,E2 -15641.062} C_VEL
LIN {X 0,Y 323.452,Z 869.293,A -85,B 0,C 180,E1 -15642.29,E2 -15642.29} C_VEL
LIN {X 0,Y 321.787,Z 876.757,A -85,B 0,C 180,E1 -15643.864,E2 -15643.864} C_VEL
LIN {X 0,Y 320.353,Z 882.686,A -85,B 0,C 180,E1 -15645.387,E2 -15645.387} C_VEL
LIN {X 0,Y 319.309,Z 886.856,A -85,B 0,C 180,E1 -15646.638,E2 -15646.638} C_VEL
LIN {X 0,Y 317.728,Z 891.886,A -85,B 0,C 180,E1 -15648.517,E2 -15648.517} C_VEL
LIN {X 0,Y 316.51,Z 895.641,A -85,B 0,C 180,E1 -15650.414,E2 -15650.414} C_VEL
LIN {X 0,Y 315.327,Z 898.331,A -85,B 0,C 180,E1 -15652.315,E2 -15652.315} C_VEL
LIN {X 0,Y 314.802,Z 899.569,A -85,B 0,C 180,E1 -15653.591,E2 -15653.591} C_VEL
LIN {X 0,Y 313.953,Z 900.651,A -85,B 0,C 180,E1 -15656.149,E2 -15656.149} C_VEL
LIN {X 0,Y 313.538,Z 900.56,A -85,B 0,C 180,E1 -15657.431,E2 -15657.431} C_VEL
LIN {X 0,Y 313.298,Z 900.008,A -85,B 0,C 180,E1 -15658.715,E2 -15658.715} C_VEL
LIN {X 0,Y 312.905,Z 898.992,A -85,B 0,C 180,E1 -15660,E2 -15660} C_VEL
LIN {X 0,Y 312.877,Z 897.598,A -85,B 0,C 180,E1 -15661.287,E2 -15661.287} C_VEL
LIN {X 0,Y 312.617,Z 894.637,A -85,B 0,C 180,E1 -15663.222,E2 -15663.222} C_VEL
LIN {X 0,Y 312.769,Z 890.551,A -85,B 0,C 180,E1 -15665.157,E2 -15665.157} C_VEL
LIN {X 0,Y 313.186,Z 883.941,A -85,B 0,C 180,E1 -15667.488,E2 -15667.488} C_VEL
LIN {X 0,Y 313.567,Z 877.923,A -85,B 0,C 180,E1 -15669.191,E2 -15669.191} C_VEL
LIN {X 0,Y 313.864,Z 871.821,A -85,B 0,C 180,E1 -15670.646,E2 -15670.646} C_VEL
LIN {X 0,Y 314.291,Z 865.516,A -85,B 0,C 180,E1 -15671.938,E2 -15671.938} C_VEL
LIN {X 0,Y 314.859,Z 856.068,A -85,B 0,C 180,E1 -15673.555,E2 -15673.555} C_VEL
LIN {X 0,Y 315.438,Z 847.033,A -85,B 0,C 180,E1 -15674.846,E2 -15674.846} C_VEL
LIN {X 0,Y 316.04,Z 837.622,A -85,B 0,C 180,E1 -15675.974,E2 -15675.974} C_VEL
LIN {X 0,Y 316.529,Z 828.124,A -85,B 0,C 180,E1 -15676.925,E2 -15676.925} C_VEL
LIN {X 0,Y 316.948,Z 818.622,A -85,B 0,C 180,E1 -15677.713,E2 -15677.713} C_VEL
LIN {X 0,Y 317.27,Z 808.39,A -85,B 0,C 180,E1 -15678.401,E2 -15678.401} C_VEL
LIN {X 0,Y 317.519,Z 797.297,A -85,B 0,C 180,E1 -15678.971,E2 -15678.971} C_VEL
LIN {X 0,Y 317.725,Z 782.816,A -85,B 0,C 180,E1 -15679.495,E2 -15679.495} C_VEL
LIN {X 0,Y 318.899,Z 733.67,A -85,B 0,C 180,E1 -15681.003,E2 -15681.003} C_VEL
LIN {X 0,Y 312.583,Z 713.545,A -85,B 0,C 180,E1 -15681.955,E2 -15681.955} C_VEL
LIN {X 0,Y 312.553,Z 713.55,A -85,B 0,C 180,E1 -15685.905,E2 -15685.905} C_VEL
LIN {X 0,Y 312.495,Z 713.557,A -85,B 0,C 180,E1 -15689.655,E2 -15689.655} C_VEL
LIN {X 0,Y 312.542,Z 713.549,A -85,B 0,C 180,E1 -15693.686,E2 -15693.686} C_VEL
LIN {X 0,Y 312.531,Z 713.553,A -85,B 0,C 180,E1 -15697.385,E2 -15697.385} C_VEL
LIN {X 0,Y 312.462,Z 713.562,A -85,B 0,C 180,E1 -15700.714,E2 -15700.714} C_VEL
LIN {X 0,Y 312.471,Z 713.554,A -85,B 0,C 180,E1 -15704.207,E2 -15704.207} C_VEL
LIN {X 0,Y 312.474,Z 713.555,A -85,B 0,C 180,E1 -15707.921,E2 -15707.921} C_VEL
LIN {X 0,Y 312.495,Z 713.552,A -85,B 0,C 180,E1 -15711.92,E2 -15711.92} C_VEL
LIN {X 0,Y 312.549,Z 713.546,A -85,B 0,C 180,E1 -15714.215,E2 -15714.215} C_VEL
LIN {X 0,Y 312.518,Z 713.551,A -85,B 0,C 180,E1 -15717.328,E2 -15717.328} C_VEL
LIN {X 0,Y 312.5,Z 713.556,A -85,B 0,C 180,E1 -15721.295,E2 -15721.295} C_VEL
LIN {X 0,Y 312.539,Z 713.552,A -85,B 0,C 180,E1 -15724.579,E2 -15724.579} C_VEL
LIN {X 0,Y 313.652,Z 716.598,A -85,B 0,C 180,E1 -15724.762,E2 -15724.762} C_VEL
LIN {X 0,Y 322.664,Z 735.813,A -85,B 0,C 180,E1 -15726.012,E2 -15726.012} C_VEL
LIN {X 0,Y 324.845,Z 741.001,A -85,B 0,C 180,E1 -15726.316,E2 -15726.316} C_VEL
LIN {X 0,Y 324.059,Z 789.617,A -85,B 0,C 180,E1 -15727.409,E2 -15727.409} C_VEL
LIN {X 0,Y 323.977,Z 802.825,A -85,B 0,C 180,E1 -15727.82,E2 -15727.82} C_VEL
LIN {X 0,Y 323.578,Z 815.885,A -85,B 0,C 180,E1 -15728.492,E2 -15728.492} C_VEL
LIN {X 0,Y 322.822,Z 827.416,A -85,B 0,C 180,E1 -15729.308,E2 -15729.308} C_VEL
LIN {X 0,Y 321.834,Z 838.998,A -85,B 0,C 180,E1 -15730.386,E2 -15730.386} C_VEL
LIN {X 0,Y 320.658,Z 849.468,A -85,B 0,C 180,E1 -15731.628,E2 -15731.628} C_VEL
LIN {X 0,Y 319.418,Z 859.067,A -85,B 0,C 180,E1 -15733.043,E2 -15733.043} C_VEL
LIN {X 0,Y 318.297,Z 867.762,A -85,B 0,C 180,E1 -15734.628,E2 -15734.628} C_VEL
LIN {X 0,Y 316.883,Z 876.266,A -85,B 0,C 180,E1 -15736.526,E2 -15736.526} C_VEL
LIN {X 0,Y 315.693,Z 883.029,A -85,B 0,C 180,E1 -15738.434,E2 -15738.434} C_VEL
LIN {X 0,Y 314.999,Z 888.395,A -85,B 0,C 180,E1 -15740.359,E2 -15740.359} C_VEL
LIN {X 0,Y 314.538,Z 891.331,A -85,B 0,C 180,E1 -15741.641,E2 -15741.641} C_VEL
LIN {X 0,Y 313.638,Z 894.892,A -85,B 0,C 180,E1 -15743.559,E2 -15743.559} C_VEL
LIN {X 0,Y 313.289,Z 896.715,A -85,B 0,C 180,E1 -15744.844,E2 -15744.844} C_VEL
LIN {X 0,Y 313.098,Z 899.028,A -85,B 0,C 180,E1 -15747.419,E2 -15747.419} C_VEL
LIN {X 0,Y 312.884,Z 899.87,A -85,B 0,C 180,E1 -15749.991,E2 -15749.991} C_VEL
LIN {X 0,Y 313.099,Z 899.106,A -85,B 0,C 180,E1 -15752.564,E2 -15752.564} C_VEL
LIN {X 0,Y 313.271,Z 896.876,A -85,B 0,C 180,E1 -15755.14,E2 -15755.14} C_VEL
LIN {X 0,Y 313.864,Z 894.06,A -85,B 0,C 180,E1 -15757.065,E2 -15757.065} C_VEL
LIN {X 0,Y 314.692,Z 890.233,A -85,B 0,C 180,E1 -15758.985,E2 -15758.985} C_VEL
LIN {X 0,Y 315.504,Z 884.761,A -85,B 0,C 180,E1 -15761.107,E2 -15761.107} C_VEL
LIN {X 0,Y 316.641,Z 877.948,A -85,B 0,C 180,E1 -15763.141,E2 -15763.141} C_VEL
LIN {X 0,Y 317.996,Z 869.92,A -85,B 0,C 180,E1 -15765.042,E2 -15765.042} C_VEL
LIN {X 0,Y 319.168,Z 861.702,A -85,B 0,C 180,E1 -15766.624,E2 -15766.624} C_VEL
LIN {X 0,Y 320.434,Z 851.532,A -85,B 0,C 180,E1 -15768.202,E2 -15768.202} C_VEL
LIN {X 0,Y 321.701,Z 841.064,A -85,B 0,C 180,E1 -15769.493,E2 -15769.493} C_VEL
LIN {X 0,Y 322.802,Z 829.268,A -85,B 0,C 180,E1 -15770.646,E2 -15770.646} C_VEL
LIN {X 0,Y 323.627,Z 816.72,A -85,B 0,C 180,E1 -15771.562,E2 -15771.562} C_VEL
LIN {X 0,Y 324.004,Z 805.29,A -85,B 0,C 180,E1 -15772.177,E2 -15772.177} C_VEL
LIN {X 0,Y 324.131,Z 794.866,A -85,B 0,C 180,E1 -15772.561,E2 -15772.561} C_VEL
LIN {X 0,Y 324.658,Z 753.877,A -85,B 0,C 180,E1 -15773.506,E2 -15773.506} C_VEL
LIN {X 0,Y 324.88,Z 741.013,A -85,B 0,C 180,E1 -15773.795,E2 -15773.795} C_VEL
LIN {X 0,Y 316.235,Z 721.791,A -85,B 0,C 180,E1 -15774.995,E2 -15774.995} C_VEL
LIN {X 0,Y 312.666,Z 714.078,A -85,B 0,C 180,E1 -15775.507,E2 -15775.507} C_VEL
LIN {X 0,Y 312.586,Z 713.542,A -85,B 0,C 180,E1 -15775.546,E2 -15775.546} C_VEL
LIN {X 0,Y 312.511,Z 713.553,A -85,B 0,C 180,E1 -15779.641,E2 -15779.641} C_VEL
LIN {X 0,Y 312.48,Z 713.556,A -85,B 0,C 180,E1 -15780.183,E2 -15780.183} C_VEL
LIN {X 0,Y 311.788,Z 713.648,A -85,B 0,C 180,E1 -15781.259,E2 -15781.259} C_VEL
LIN {X 0,Y 308.911,Z 714.007,A -85,B 0,C 180,E1 -15783.011,E2 -15783.011} C_VEL
LIN {X 0,Y 306.504,Z 714.304,A -85,B 0,C 180,E1 -15784.432,E2 -15784.432} C_VEL
LIN {X 0,Y 305.502,Z 714.434,A -85,B 0,C 180,E1 -15785.532,E2 -15785.532} C_VEL
LIN {X 0,Y 305.435,Z 714.436,A -85,B 0,C 180,E1 -15785.905,E2 -15785.905} C_VEL
LIN {X 0,Y 305.446,Z 714.418,A -85,B 0,C 180,E1 -15788.528,E2 -15788.528} C_VEL
LIN {X 0,Y 305.481,Z 714.434,A -85,B 0,C 180,E1 -15792.591,E2 -15792.591} C_VEL
LIN {X 0,Y 305.489,Z 714.416,A -85,B 0,C 180,E1 -15796.356,E2 -15796.356} C_VEL
LIN {X 0,Y 305.436,Z 714.439,A -85,B 0,C 180,E1 -15799.889,E2 -15799.889} C_VEL
LIN {X 0,Y 305.448,Z 714.439,A -85,B 0,C 180,E1 -15803.62,E2 -15803.62} C_VEL
LIN {X 0,Y 305.412,Z 714.436,A -85,B 0,C 180,E1 -15806.476,E2 -15806.476} C_VEL
LIN {X 0,Y 305.41,Z 714.44,A -85,B 0,C 180,E1 -15809.585,E2 -15809.585} C_VEL
LIN {X 0,Y 305.462,Z 714.435,A -85,B 0,C 180,E1 -15812.603,E2 -15812.603} C_VEL
LIN {X 0,Y 305.447,Z 714.431,A -85,B 0,C 180,E1 -15815.533,E2 -15815.533} C_VEL
LIN {X 0,Y 305.456,Z 714.435,A -85,B 0,C 180,E1 -15819.81,E2 -15819.81} C_VEL
LIN {X 0,Y 305.509,Z 714.417,A -85,B 0,C 180,E1 -15822.599,E2 -15822.599} C_VEL
LIN {X 0,Y 305.583,Z 714.419,A -85,B 0,C 180,E1 -15825.346,E2 -15825.346} C_VEL
LIN {X 0,Y 305.572,Z 714.408,A -85,B 0,C 180,E1 -15829.397,E2 -15829.397} C_VEL
LIN {X 0,Y 305.736,Z 714.402,A -85,B 0,C 180,E1 -15832.072,E2 -15832.072} C_VEL
LIN {X 0,Y 305.625,Z 714.411,A -85,B 0,C 180,E1 -15834.722,E2 -15834.722} C_VEL
LIN {X 0,Y 305.894,Z 714.384,A -85,B 0,C 180,E1 -15838.683,E2 -15838.683} C_VEL
LIN {X 0,Y 305.894,Z 714.377,A -85,B 0,C 180,E1 -15841.316,E2 -15841.316} C_VEL
LIN {X 0,Y 305.626,Z 714.419,A -85,B 0,C 180,E1 -15845.278,E2 -15845.278} C_VEL
LIN {X 0,Y 305.736,Z 714.396,A -85,B 0,C 180,E1 -15847.928,E2 -15847.928} C_VEL
LIN {X 0,Y 305.538,Z 714.427,A -85,B 0,C 180,E1 -15851.948,E2 -15851.948} C_VEL
LIN {X 0,Y 305.572,Z 714.422,A -85,B 0,C 180,E1 -15855.037,E2 -15855.037} C_VEL
LIN {X 0,Y 305.515,Z 714.427,A -85,B 0,C 180,E1 -15858.787,E2 -15858.787} C_VEL
LIN {X 0,Y 305.426,Z 714.437,A -85,B 0,C 180,E1 -15863.044,E2 -15863.044} C_VEL
LIN {X 0,Y 305.466,Z 714.425,A -85,B 0,C 180,E1 -15866.224,E2 -15866.224} C_VEL
LIN {X 0,Y 305.438,Z 714.435,A -85,B 0,C 180,E1 -15869.056,E2 -15869.056} C_VEL
LIN {X 0,Y 305.392,Z 714.443,A -85,B 0,C 180,E1 -15871.958,E2 -15871.958} C_VEL
LIN {X 0,Y 305.41,Z 714.439,A -85,B 0,C 180,E1 -15875.12,E2 -15875.12} C_VEL
LIN {X 0,Y 305.433,Z 714.419,A -85,B 0,C 180,E1 -15878.544,E2 -15878.544} C_VEL
LIN {X 0,Y 305.476,Z 714.432,A -85,B 0,C 180,E1 -15882.607,E2 -15882.607} C_VEL
LIN {X 0,Y 305.492,Z 714.429,A -85,B 0,C 180,E1 -15886.373,E2 -15886.373} C_VEL
LIN {X 0,Y 305.478,Z 714.55,A -85,B 0,C 180,E1 -15890.412,E2 -15890.412} C_VEL
LIN {X 0,Y 309.054,Z 728.234,A -85,B 0,C 180,E1 -15894.084,E2 -15894.084} C_VEL
LIN {X 0,Y 311.597,Z 739.526,A -85,B 0,C 180,E1 -15896.909,E2 -15896.909} C_VEL
LIN {X 0,Y 313.25,Z 748.063,A -85,B 0,C 180,E1 -15898.947,E2 -15898.947} C_VEL
LIN {X 0,Y 310.112,Z 770.263,A -85,B 0,C 180,E1 -15903.62,E2 -15903.62} C_VEL
LIN {X 0,Y 310.101,Z 771.129,A -85,B 0,C 180,E1 -15903.736,E2 -15903.736} C_VEL
LIN {X 0,Y 314.248,Z 804.969,A -85,B 0,C 180,E1 -15904.925,E2 -15904.925} C_VEL
LIN {X 0,Y 316.75,Z 833.49,A -85,B 0,C 180,E1 -15905.818,E2 -15905.818} C_VEL
LIN {X 0,Y 315.451,Z 882.212,A -85,B 0,C 180,E1 -15906.933,E2 -15906.933} C_VEL
LIN {X 0,Y 314.632,Z 895.368,A -85,B 0,C 180,E1 -15907.477,E2 -15907.477} C_VEL
LIN {X 0,Y 313.292,Z 908.617,A -85,B 0,C 180,E1 -15908.286,E2 -15908.286} C_VEL
LIN {X 0,Y 311.887,Z 919.794,A -85,B 0,C 180,E1 -15909.223,E2 -15909.223} C_VEL
LIN {X 0,Y 310.226,Z 931.463,A -85,B 0,C 180,E1 -15910.49,E2 -15910.49} C_VEL
LIN {X 0,Y 308.607,Z 942.003,A -85,B 0,C 180,E1 -15911.934,E2 -15911.934} C_VEL
LIN {X 0,Y 307.373,Z 950.676,A -85,B 0,C 180,E1 -15913.403,E2 -15913.403} C_VEL
LIN {X 0,Y 306.236,Z 958.561,A -85,B 0,C 180,E1 -15915.016,E2 -15915.016} C_VEL
LIN {X 0,Y 305.247,Z 966.594,A -85,B 0,C 180,E1 -15917.037,E2 -15917.037} C_VEL
LIN {X 0,Y 304.581,Z 973.918,A -85,B 0,C 180,E1 -15919.372,E2 -15919.372} C_VEL
LIN {X 0,Y 304.438,Z 978.844,A -85,B 0,C 180,E1 -15921.379,E2 -15921.379} C_VEL
LIN {X 0,Y 304.542,Z 982.646,A -85,B 0,C 180,E1 -15923.383,E2 -15923.383} C_VEL
LIN {X 0,Y 304.657,Z 984.615,A -85,B 0,C 180,E1 -15924.715,E2 -15924.715} C_VEL
LIN {X 0,Y 304.872,Z 986.108,A -85,B 0,C 180,E1 -15926.043,E2 -15926.043} C_VEL
LIN {X 0,Y 304.925,Z 987.158,A -85,B 0,C 180,E1 -15927.367,E2 -15927.367} C_VEL
LIN {X 0,Y 305.036,Z 987.808,A -85,B 0,C 180,E1 -15928.689,E2 -15928.689} C_VEL
LIN {X 0,Y 305.144,Z 988.044,A -85,B 0,C 180,E1 -15930.009,E2 -15930.009} C_VEL
LIN {X 0,Y 305.036,Z 987.795,A -85,B 0,C 180,E1 -15931.329,E2 -15931.329} C_VEL
LIN {X 0,Y 304.926,Z 987.136,A -85,B 0,C 180,E1 -15932.651,E2 -15932.651} C_VEL
LIN {X 0,Y 304.869,Z 986.075,A -85,B 0,C 180,E1 -15933.974,E2 -15933.974} C_VEL
LIN {X 0,Y 304.638,Z 984.565,A -85,B 0,C 180,E1 -15935.303,E2 -15935.303} C_VEL
LIN {X 0,Y 304.475,Z 981.961,A -85,B 0,C 180,E1 -15937.002,E2 -15937.002} C_VEL
LIN {X 0,Y 304.462,Z 977.27,A -85,B 0,C 180,E1 -15939.307,E2 -15939.307} C_VEL
LIN {X 0,Y 305.156,Z 968.218,A -85,B 0,C 180,E1 -15942.646,E2 -15942.646} C_VEL
LIN {X 0,Y 306.045,Z 961.373,A -85,B 0,C 180,E1 -15944.64,E2 -15944.64} C_VEL
LIN {X 0,Y 306.727,Z 956.828,A -85,B 0,C 180,E1 -15945.773,E2 -15945.773} C_VEL
LIN {X 0,Y 308.554,Z 946.679,A -85,B 0,C 180,E1 -15947.916,E2 -15947.916} C_VEL
LIN {X 0,Y 310.614,Z 936.107,A -85,B 0,C 180,E1 -15949.675,E2 -15949.675} C_VEL
LIN {X 0,Y 312.515,Z 927.074,A -85,B 0,C 180,E1 -15950.924,E2 -15950.924} C_VEL
LIN {X 0,Y 314.31,Z 917.816,A -85,B 0,C 180,E1 -15952.003,E2 -15952.003} C_VEL
LIN {X 0,Y 316.342,Z 906.694,A -85,B 0,C 180,E1 -15953.059,E2 -15953.059} C_VEL
LIN {X 0,Y 318.343,Z 895.035,A -85,B 0,C 180,E1 -15953.94,E2 -15953.94} C_VEL
LIN {X 0,Y 319.851,Z 884.211,A -85,B 0,C 180,E1 -15954.596,E2 -15954.596} C_VEL
LIN {X 0,Y 321.114,Z 873.363,A -85,B 0,C 180,E1 -15955.098,E2 -15955.098} C_VEL
LIN {X 0,Y 324.202,Z 833.554,A -85,B 0,C 180,E1 -15956.586,E2 -15956.586} C_VEL
LIN {X 0,Y 323.962,Z 809.404,A -85,B 0,C 180,E1 -15957.879,E2 -15957.879} C_VEL
LIN {X 0,Y 322.812,Z 790.691,A -85,B 0,C 180,E1 -15959.146,E2 -15959.146} C_VEL
LIN {X 0,Y 321.345,Z 774.258,A -85,B 0,C 180,E1 -15960.447,E2 -15960.447} C_VEL
LIN {X 0,Y 320.174,Z 763.031,A -85,B 0,C 180,E1 -15961.447,E2 -15961.447} C_VEL
LIN {X 0,Y 319.302,Z 755.411,A -85,B 0,C 180,E1 -15962.181,E2 -15962.181} C_VEL
